// POUs/[Internal]/Beta Function Blocks/Position Correction/MC_TableBasedPositionCompensation
(*==============================================================================*)
(* Name:	MC_TableBasedPositionCompensation									*)
(*		(based on _FB_PositionCorrectionTableLookup + MC_PositionCorrectionLimiter)	*)
(* Parameter: returns a compensation value depending on the position of the reference axis	*)
(*		Use the nc function PositionCompensation to compensate a position error	*)
(*		1. the FB _FB_PositionCorrectionTableLookup calculates the correction value	*)
(*		2. the FB MC_PositionCorrectionLimiter feed this correction value		*)
(*		into the NcToPlc.PositionCorrection variable							*)
(* Author:	 	HKP																*)
(* Date:		19-July-2012													*)
(* last edit:	VER 0.0.4														*)
(*==============================================================================*)
FUNCTION_BLOCK MC_TableBasedPositionCompensation
VAR_IN_OUT
	Axis						: AXIS_REF; (*Reference to an axis*)
END_VAR
VAR_INPUT
	Enable						: BOOL; 				(* rising edge triggers initialize routine *)
	pTable						: POINTER TO ST_PositionCompensationTableElement;	(* pointer to equidistant table with strictly monotonous increasing position values *)
	TableSize					: UDINT;				(* size of data in bytes related to 'pTable' *)
	TableParameter				: ST_PositionCompensationTableParameter;(* position compensation table parameter structure *)
	Ramp						: LREAL;								(* velocity limit for feeded position compensation (constant velocity and linear position sub profile for position compensation) [mm/s] (default:=0.0) *)
	DisableMode					: E_DisableMode;						(* disable mode defines whow to react in case of disabling: (0)=HOLD, (1)=RESET, ... *)
	Options						: ST_PositionCompensationOptions;		(* optional parameters (NOT USED YET) *)
END_VAR
VAR_OUTPUT
	Enabled						: BOOL;
	Busy						: BOOL;
	Error						: BOOL;
{attribute 'displaymode':='hex'}
	ErrorID						: UDINT;
	CurrentCorrection			: LREAL;							(* current actual position correction value [mm] *)
	Limiting					: BOOL;								(* function block is currently limiting the Position Correction *)
END_VAR
VAR
	InternalEnable				: BOOL;								(* trick for internal FB handling *)
	state						: INT;
	GetThisTaskIndex			: GETCURTASKINDEX;
	CycleTime					: LREAL;							(* task cycle time [s] *)
	fbCalcPositionCorrection	: _FB_PositionCorrectionTableLookup;(* based on old 'FB_PositionCompensation' in TcNc.lib *)
	fbFeedPositionCorrection	: MC_PositionCorrectionLimiter;		(* s.TcMC2.lib (original based on old 'FB_WritePositionCorrection' in TcNc.lib) *)
	CalcPosCorrOut				: ST_McOutputs;
	FeedPosCorrOut				: ST_McOutputs;
	InternalAcceleration		: LREAL;							(* input of FB 'MC_PositionCorrectionLimiter': 'Acceleration' [mm/s^2] *)
	InternalCorrectionValue		: LREAL;							(* output of FB 'MC_PositionCorrectionLimiter': 'PositionCorrectionValue' [mm] *)
	InternalLimitingActive		: BOOL;								(* output of FB 'MC_PositionCorrectionLimiter': 'Limiting' [0/1] *)
END_VAR


CASE state OF
	0 : (* init *)
		Busy := FALSE;
		Enabled := FALSE;
		IF Enable THEN
			IF NOT Axis.NcToPlc.OpModeDWord.20 THEN (* PositionCorrection active ? *)
				Error := TRUE;
				ErrorID := MC_ERROR_WRONG_MODE;
				state := 9999;
			ELSIF Ramp < 0 THEN
				Error := TRUE;
				ErrorID := MC_ERROR_PARAMETER_NOT_CORRECT;
				state := 9999;
			ELSE
				Busy := TRUE;
				state := 1;
			END_IF
		END_IF

	1 : (* active *)
		Enabled := TRUE;


		(* cycle time needed for pre calculation of the acceleration input *)
		IF CycleTime = 0 THEN
			GetThisTaskIndex();
(*			CycleTime := SystemTaskInfoArr[GetThisTaskIndex.index].cycleTime * LREAL#100E-9;*)
			CycleTime := TwinCAT_SystemInfoVarList._TaskInfo[GetThisTaskIndex.index].cycleTime * LREAL#100E-9;
		END_IF

		(* special handling for disabling (depends from disable mode) *)
		IF( Enable = FALSE ) THEN
			(* disable mode HOLD *)
			IF( (DisableMode = DisableModeHold) ) THEN
				InternalEnable := TRUE;
				IF( Ramp > 0.0 ) THEN
					InternalAcceleration := Ramp / CycleTime;			(* mm/s^2 = mm/s / s *)
				ELSE
					InternalAcceleration := 0.0;
				END_IF
			(* disable mode RESET *)
			ELSE
				InternalEnable := Enable;
				InternalAcceleration := 0.0;
			END_IF
		(* active *)
		ELSE
			InternalEnable := Enable;
			IF( Ramp > 0.0 ) THEN
				InternalAcceleration := Ramp / CycleTime;			(* mm/s^2 = mm/s / s *)
			ELSE
				InternalAcceleration := 0.0;
			END_IF
		END_IF


		(* 1.) calculate position correction (if enabled) *)
		(* '_FB_PositionCorrectionTableLookup' *)
		fbCalcPositionCorrection(
		   (* Enable := Enable, *)
		   Enable := InternalEnable,
		   pTable := pTable,
		   TableSize := TableSize,
		   Axis := Axis,
		   TableParameter := TableParameter,
		   Compensation => InternalCorrectionValue,
		   Error => CalcPosCorrOut.Error,
		   ErrorId => CalcPosCorrOut.ErrorID,
		   Active => CalcPosCorrOut.Active );

		(* check for error return code *)
		IF CalcPosCorrOut.Error THEN
			Error := TRUE;
			ErrorID := CalcPosCorrOut.ErrorID;
			state := 9999;
		END_IF


		(* 2.) feed position compensation (acceleration limited, that means linear velocity ramp) *)
		(*
				POSITIONCORRECTIONMODE_FAST
					The limitatation to maximum position change per cycle. Due to the maximum 
					change per cycle, the correction will take place as fast as possible and may 
					also be unlimited if PositionCorrectionValue is changed slightly. 
		*)
		(* MC_PositionCorrectionLimiter *)
		fbFeedPositionCorrection(
		(*	Enable :=TRUE, *)
			 Enable :=Enable,
			 PositionCorrectionValue := InternalCorrectionValue,
			 CorrectionMode := POSITIONCORRECTION_MODE_FAST,
			 Acceleration := InternalAcceleration,			(* HKP: pre calculated internal acceleration limit *)
			 CorrectionLength := 0.0,					(* optional length - not used for this correction mode 'POSITIONCORRECTION_MODE_FAST' *)
			 Axis := Axis,
			 Busy => FeedPosCorrOut.Busy,
			 Error => FeedPosCorrOut.Error,
			 ErrorID =>FeedPosCorrOut.ErrorID,
			 Limiting => InternalLimitingActive
			);

		(* check for error return code *)
		IF FeedPosCorrOut.Error THEN
			Error := TRUE;
			ErrorID := FeedPosCorrOut.ErrorID;
			state := 9999;
		END_IF


		CurrentCorrection	:= InternalCorrectionValue;
		Limiting			:= InternalLimitingActive;

		IF NOT Enable THEN
			Enabled := FALSE;
			state := 0;
		END_IF

	9999 : (* error *)
		IF NOT Enable THEN
			Error := FALSE;
			ErrorID := 0;
			state := 0;
		END_IF
END_CASE

IF state = 0 THEN
	Busy := FALSE;
END_IF

END_FUNCTION_BLOCK

// POUs/[Internal]/_FB_PositionCorrectionTableLookup
{attribute 'conditionalshow'}
(*==========================================================================*)
(* Name:	_FB_PositionCorrectionTableLookup (based on FB_PositionCompensation)	*)
(* Parameter:	returns a compensation value depending on the position of the reference	*)
(*			axis																*)
(*																			*)
(* Author:	 	kbn & HKP														*)
(* Date:		06-July-2012														*)
(* last edit:	VER 2.0.0														*)
(*==========================================================================*)
FUNCTION_BLOCK _FB_PositionCorrectionTableLookup
VAR_IN_OUT
	Axis				: AXIS_REF; (*Reference to an axis*)
END_VAR
VAR_INPUT
	Enable			: BOOL; 				(* rising edge triggers initialize routine *)
	pTable			: POINTER TO ST_PositionCompensationTableElement;	(* pointer to table of this type *)
	TableSize		: UDINT;				(* size of data in bytes related to 'pTable' *)
	TableParameter	: ST_PositionCompensationTableParameter;	(* position compensation table parameter structure *)
END_VAR
VAR_OUTPUT
	Compensation	: LREAL;
	Error			: BOOL;
{attribute 'displaymode':='hex'}
	ErrorID			: UDINT;
	Active			: BOOL;
END_VAR
VAR
	nState			: UDINT;
	dwSize			: DWORD;
	eActiveDirection	: E_WorkDirection := WorkDirectionNone;
	bExecCalc		: BOOL;
	stElement1		: ST_PositionCompensationTableElement;
	stElement2		: ST_PositionCompensationTableElement;
	nLeftIndex		: UDINT;									(* Index starting from 0 up to (N-1) *)
	fSetPos			: LREAL;									(* position setpoint (absolute linear position or modulo position) *)
	(* HKP *)
	pTmpTable		: POINTER TO ST_PositionCompensationTableElement;	(* helper variable: pointer to table of this type *)
	fTmpStep		: LREAL;									(* helper variable *)
	fTmpA			: LREAL;									(* helper variable *)
	fTmpB			: LREAL;									(* helper variable *)
	fTmpDelta1		: LREAL;									(* helper variable *)
	fTmpDelta2		: LREAL;									(* helper variable *)
END_VAR
VAR CONSTANT
	ERRORCODE_PARAMSIZE	: UDINT := 16#4B43;
	ERRORCODE_PARAMPOS	: UDINT := 16#4B44;
(*	ERRORCODE_TCNCNOTIMPL	: UDINT := 16#4B45; *)
END_VAR

(* get last commanded direction *)
IF Axis.NcToPlc.SetVelo > 0.0001 THEN
	eActiveDirection	:= WorkDirectionPositive;
ELSIF Axis.NcToPlc.SetVelo < -0.0001 THEN
	eActiveDirection	:= WorkDirectionNegative;
END_IF

CASE nState OF
0:
	Error			:= FALSE;
	ErrorId			:= 0;
	Compensation	:= 0.0;
	Active			:= FALSE;
	bExecCalc		:= FALSE;

	IF Enable THEN
		(* reinitialize *)
		IF ( ABS(Axis.NcToPlc.SetVelo) < 0.0001 ) THEN
			eActiveDirection := WorkDirectionNone;
		END_IF
		(* check table size (in mimimum 2 elements needed) *)
		IF TableParameter.NoOfTableElements < 2 THEN
			Error	:= TRUE;
			ErrorId	:= ERRORCODE_PARAMSIZE;
			nState	:= 9999;
			RETURN;
		END_IF
		(* check table size *)
		IF TableParameter.NoOfTableElements*SIZEOF(pTable^) <> TableSize THEN
			Error	:= TRUE;
			ErrorId	:= ERRORCODE_PARAMSIZE;
			nState	:= 9999;
			RETURN;
		END_IF
		(* ====================================================== *)
		(* HKP: read table element with index (0)						*)
		(* ====================================================== *)
		(* stElement1	:= F_GetCompensationElementAt(pTable:=pTable, nElement:=0); *)
		pTmpTable	:= pTable + (SIZEOF(pTable^) * (UDINT#0));
		stElement1	:= pTmpTable^;
		(* ====================================================== *)
		IF stElement1.Position <> TableParameter.MinPosition THEN
			Error	:= TRUE;
			ErrorId	:= ERRORCODE_PARAMPOS;
			nState	:= 9999;
			RETURN;
		END_IF
		(* ====================================================== *)
		(* HKP: read table element with index (Parameter.nTableElements-1)	*)
		(* ====================================================== *)
		(* stElement1	:= F_GetCompensationElementAt(pTable:=pTable, nElement:=Parameter.nTableElements-1); *)
		pTmpTable	:= pTable + (SIZEOF(pTable^) * (TableParameter.NoOfTableElements-1));
		stElement1	:= pTmpTable^;
		(* ====================================================== *)
		IF stElement1.Position <> TableParameter.MaxPosition THEN
			Error	:= TRUE;
			ErrorId	:= ERRORCODE_PARAMPOS;
			nState	:= 9999;
			RETURN;
		END_IF
		(* HKP: This two parameter are not needed yet *)
		(* IF Parameter.eTableType <> TableType1DEquidistant OR Parameter.bModulo THEN
			Error	:= TRUE;
			ErrorId	:= ERRORCODE_TCNCNOTIMPL;
			nState	:= 9999;
			RETURN;
		END_IF *)

		(* check for equidistant table (table must contain in minimum 2 elements) *)
		pTmpTable	:= pTable + (SIZEOF(pTable^) * (UDINT#1));						(* read index 1 *)
		stElement2	:= pTmpTable^;
		pTmpTable	:= pTable + (SIZEOF(pTable^) * (UDINT#0));						(* read index 0 *)
		stElement1	:= pTmpTable^;
		fTmpDelta1	:= stElement2.Position - stElement1.Position;						(* calculate position delta 1: (index 1 - index 0) *)
		pTmpTable	:= pTable + (SIZEOF(pTable^) * (TableParameter.NoOfTableElements-1));	(* read index (n) *)
		stElement2	:= pTmpTable^;
		pTmpTable	:= pTable + (SIZEOF(pTable^) * (TableParameter.NoOfTableElements-2));	(* read index (n-1) *)
		stElement1	:= pTmpTable^;
		fTmpDelta2	:= stElement2.Position - stElement1.Position;						(* calculate position delta 2: (index (n) - index (n-1)) *)
		IF( ABS(fTmpDelta2 - fTmpDelta1) > 1.0E-6 ) THEN
			Error	:= TRUE;
			ErrorId	:= ERRORCODE_PARAMPOS;
			nState	:= 9999;
			RETURN;
		END_IF

		(* ====================================================== *)
		(* HKP: call action 'F_IsCompensationDirection()'				*)
		(* INPUT: eActive:=eActiveDirection, eRequested:=Parameter.Direction *)
		(* OUTPUT: bExecCalc									*)
		(* ====================================================== *)
		(* bExecCalc	:= F_IsCompensationDirection(eActive:=eActiveDirection, eRequested:=Parameter.Direction); *)
		ActIsCompensationDirection( );
		(* ====================================================== *)
		nState	:= 10;
	END_IF
10:
	(* ====================================================== *)
	(* HKP: call action 'F_IsCompensationDirection()'				*)
	(* INPUT: eActive:=eActiveDirection, eRequested:=Parameter.Direction *)
	(* OUTPUT: bExecCalc									*)
	(* ====================================================== *)
	(* bExecCalc	:= F_IsCompensationDirection(eActive:=eActiveDirection, eRequested:=Parameter.Direction); *)
	ActIsCompensationDirection( );
	(* ====================================================== *)
	IF NOT Enable THEN
		bExecCalc	:= FALSE;
		nState		:= 0;
	END_IF


9999:
	IF NOT Enable THEN
		nState	:= 0;
	END_IF

END_CASE


IF bExecCalc THEN
	(* compensation is generally enabled & direction is ok *)
	Active	:= TRUE;
	(* modulo or linear axis? *)
	IF( TableParameter.Modulo )THEN
		fSetPos	:= Axis.NcToPlc.ModuloSetPos;
	ELSE
		fSetPos	:= Axis.NcToPlc.SetPos;
	END_IF
	IF fSetPos < TableParameter.MinPosition THEN
		(* ====================================================== *)
		(* HKP: read table element with index (0)						*)
		(* ====================================================== *)
		(* stElement1	:= F_GetCompensationElementAt(pTable:=pTable, nElement:=0 ); *)
		pTmpTable	:= pTable + (SIZEOF(pTable^) * (UDINT#0));
		stElement1	:= pTmpTable^;
		(* ====================================================== *)
		Compensation	:= stElement1.Compensation;
	ELSIF fSetPos > TableParameter.MaxPosition THEN
		(* ====================================================== *)
		(* HKP: read table element with index (Parameter.nTableElements-1)	*)
		(* ====================================================== *)
		(* stElement1	:= F_GetCompensationElementAt(pTable:=pTable, nElement:=Parameter.nTableElements-1); *)
		pTmpTable	:= pTable + (SIZEOF(pTable^) * (TableParameter.NoOfTableElements-1));
		stElement1	:= pTmpTable^;
		(* ====================================================== *)
		Compensation := stElement1.Compensation;
	ELSE
		(* ====================================================== *)
		(* HKP: get left table index to position (Axis.NcToPlc.SetPos)		*)
		(* ====================================================== *)
		(* nLeftIndex	:= F_GetLeftIndex(fPos:=Axis.NcToPlc.SetPos, fMin:=Parameter.MinPosition, fMax:=Parameter.MaxPosition, nCount:=Parameter.NoOfTableElements); *)
		IF TableParameter.NoOfTableElements <= 1 THEN
			nLeftIndex := 0;
		ELSE
			IF fSetPos < TableParameter.MinPosition THEN
				nLeftIndex	:= 0;
			ELSIF fSetPos > TableParameter.MaxPosition THEN
				nLeftIndex	:= TableParameter.NoOfTableElements-1;
			ELSE
				fTmpStep	:= (TableParameter.MaxPosition-TableParameter.MinPosition)/UDINT_TO_LREAL(TableParameter.NoOfTableElements-1);
				nLeftIndex	:= LREAL_TO_UDINT(FLOOR((fSetPos-TableParameter.MinPosition)/fTmpStep));
			END_IF
		END_IF
		(* ====================================================== *)
		IF nLeftIndex >= TableParameter.NoOfTableElements-1 THEN
			(* there is no right index - probably fPos is exactly 'MaxPosition' *)
			(* ====================================================== *)
			(* HKP: read table element with index (Parameter.nTableElements-1)	*)
			(* ====================================================== *)
			(* stElement1	:= F_GetCompensationElementAt(pTable:=pTable, nElement:=Parameter.nTableElements-1); *)
			pTmpTable	:= pTable + (SIZEOF(pTable^) * (TableParameter.NoOfTableElements-1));
			stElement1	:= pTmpTable^;
			(* ====================================================== *)
			Compensation	:= stElement1.Compensation;
		ELSE
			(* ====================================================== *)
			(* HKP: read table element with index (nLeftIndex)				*)
			(* HKP: read table element with index (nLeftIndex+1)				*)
			(* ====================================================== *)
			(* stElement1	:= F_GetCompensationElementAt(pTable:=pTable, nElement:=nLeftIndex); *)
			(* stElement2	:= F_GetCompensationElementAt(pTable:=pTable, nElement:=nLeftIndex+1); *)
			pTmpTable	:= pTable + (SIZEOF(pTable^) * nLeftIndex);
			stElement1	:= pTmpTable^;
			pTmpTable	:= pTable + (SIZEOF(pTable^) * (nLeftIndex+1));
			stElement2	:= pTmpTable^;
			(* ====================================================== *)
			(* ====================================================== *)
			(* HKP: calculate linear interpolation between (stElement1) and (stElement2) for position (Axis.NcToPlc.SetPos)	*)
			(* ====================================================== *)
			(* Compensation	:= F_LinearInterpolationCompensation(fPos:=Axis.NcToPlc.SetPos, stElement1:=stElement1, stElement2:=stElement2); *)
			(* y := ax+b*)
			(* a:=(y2-y1)/(x2-x1)*)
			fTmpA	:= (stElement2.Compensation-stElement1.Compensation) / (stElement2.Position-stElement1.Position);
			(* b:=y-ax1 *)
			fTmpB	:= stElement1.Compensation - fTmpA*stElement1.Position;
			Compensation := fTmpA*fSetPos + fTmpB;
			(* ====================================================== *)
		END_IF
	END_IF
ELSE
	Compensation	:= 0.0;
	Active			:= FALSE;
END_IF

ACTION ActIsCompensationDirection:
(*
FUNCTION F_IsCompensationDirection : BOOL
VAR_INPUT
	eActiveDirection		: E_WorkingDirection;	( eActive		: E_WorkingDirection )
	Parameter.Direction	: E_WorkingDirection;	( eRequested	: E_WorkingDirection )
END_VAR
VAR_OUTPUT
	bExecCalc		: BOOL;				( F_IsCompensationDirection : BOOL )
END_VAR
*)

(*
         |Active |       |       |       |
         |None   | both  | plus  | minus |
---------|-------|-------|-------|-------|
Req None |  0    |  0    |  0    |  0    |
---------|-------|-------|-------|-------|
Req both |  1    |  d.c. |  1    |  1    |
---------|-------|-------|-------|-------|
Req plus |  0    |  0    |  1    |  0    |
---------|-------|-------|-------|-------|
Req minus|  0    |  0    |  0    |  1    |
---------|-------|-------|-------|-------|

d.c.= don't care
*)

IF TableParameter.Direction = WorkDirectionBoth THEN
	bExecCalc	:= TRUE;
	RETURN;
END_IF
IF eActiveDirection = WorkDirectionPositive AND TableParameter.Direction = WorkDirectionPositive  THEN
	bExecCalc	:= TRUE;
	RETURN;
END_IF
IF eActiveDirection = WorkDirectionNegative AND TableParameter.Direction = WorkDirectionNegative  THEN
	bExecCalc	:= TRUE;
	RETURN;
END_IF
bExecCalc		:= FALSE;


(*
IF eActiveDirection = WorkingDirectionPlus AND (TableParameter.Direction = WorkingDirectionBoth OR TableParameter.Direction = WorkingDirectionPlus ) THEN
	bExecCalc	:= TRUE;
	RETURN;
END_IF
IF eActiveDirection = WorkingDirectionMinus AND (TableParameter.Direction = WorkingDirectionBoth OR TableParameter.Direction = WorkingDirectionMinus ) THEN
	bExecCalc	:= TRUE;
	RETURN;
END_IF
bExecCalc		:= FALSE;
*)
END_ACTION

END_FUNCTION_BLOCK

// POUs/Administrative/Extensions/MC_PositionCorrectionLimiter
FUNCTION_BLOCK MC_PositionCorrectionLimiter
(*
 	The function block PositionCorrectionLimiter feed a correction value into the
	NcToPlc.PositionCorrection variable. 

	The correction value corrects the actual position of the encoder. The correction 
	does not only affect the actual position but will also lead to an axis motion caused 
	by the position controller of the axis or drive. The correction does not affect the
	set position of the set-point generator.

	The block supports following modes:
		POSITIONCORRECTIONMODE_UNLIMITED
			no limitation - the PositionCorrectionValue is passed to the NC immediately
		POSITIONCORRECTIONMODE_FAST
			The limitatation to maximum position change per cycle. Due to the maximum 
			change per cycle, the correction will take place as fast as possible and may 
			also be unlimited if PositionCorrectionValue is changed slightly. 
		POSITIONCORRECTIONMODE_FULLLENGTH 
			The limitation uses a defined full CorrectionLength (travel path)  to adapt to 
			the PositionCorrectionValue in small steps. This mode will allways cause a 
			limitation and takes care of a smooth correction.
*)
VAR_IN_OUT
	Axis					:	AXIS_REF; (*Reference to an axis*)
END_VAR
VAR_INPUT
	Enable				:	BOOL;
	PositionCorrectionValue : 	LREAL;
	CorrectionMode		:	E_AxisPositionCorrectionMode;
	Acceleration			: 	LREAL;
	CorrectionLength		:	LREAL; (* optional length - comparable to 'superposition length' *)
END_VAR
VAR_OUTPUT
	Busy				:	BOOL;
	Error				:	BOOL;
{attribute 'displaymode':='hex'}
	ErrorID				:	UDINT;
	Limiting				: 	BOOL;	(* function block is currently limiting the Position Correction *)
END_VAR
VAR
	GetThisTaskIndex: GETCURTASKINDEX;
	CycleTime: LREAL;
	MaxDeltaVelocity: LREAL;
	MaxDeltaPosition: LREAL;
	DeltaCorrection: LREAL;
	InitialDeltaCorrection: LREAL;
	EndOfEnablePhase: BOOL;
	iCorrectionMode : E_AxisPositionCorrectionMode;
	state: INT;
	NumberOfCycles: UDINT;
	DeltaCorrectionPerCycle: LREAL;
	LastPositionCorrectionValue: LREAL;
	LastPositionCorrection: LREAL;
END_VAR

CASE state OF
	0 : (* disabled *)
		Busy := FALSE;
		Limiting := FALSE;
		LastPositionCorrectionValue := 0;
		IF Enable THEN
			(* IF Acceleration<=0 AND CorrectionMode <> POSITIONCORRECTION_MODE_UNLIMITED THEN *) (* KST 20120730 *)
			IF Acceleration<0 AND CorrectionMode <> POSITIONCORRECTION_MODE_UNLIMITED THEN (* KST 20120730 - zero acc means unlimited correction *)
				Error := TRUE;
				ErrorID := MC_ERROR_PARAMETER_NOT_CORRECT;
			ELSIF CorrectionLength <= 0 AND CorrectionMode=POSITIONCORRECTION_MODE_FULLLENGTH THEN
				Error := TRUE;
				ErrorID := MC_ERROR_PARAMETER_NOT_CORRECT;
			ELSE
				Limiting := FALSE;
				Error := FALSE;
				ErrorID := 0;
				LastPositionCorrection := Axis.PlcToNc.PositionCorrection; // KST 2021-02-23 store position correction value
				state := 1;
				Busy := TRUE;
			END_IF
		ELSE
			Limiting := FALSE;
			Error := FALSE;
			ErrorID := 0;
		END_IF

	1 : (* enabled *)
		Busy := TRUE;
		IF NOT Enable THEN
			state := 2;
		END_IF

	2 : (* disabling *)
		IF Enable THEN
			LastPositionCorrection := Axis.PlcToNc.PositionCorrection; // KST 2021-09-27 store position correction value
			state := 1;
		ELSE
			PositionCorrectionValue := 0;
//			IF Axis.PlcToNc.PositionCorrection = 0 THEN
			IF LastPositionCorrection = 0 THEN	// KST 2021-02-23
				state := 0;
			END_IF
		END_IF
END_CASE

CASE state OF
	1, 2:
		IF CycleTime = 0 THEN
			GetThisTaskIndex();
			CycleTime := TwinCAT_SystemInfoVarList._TaskInfo[GetThisTaskIndex.index].cycleTime * LREAL#100E-9;
		END_IF
		MaxDeltaVelocity := Acceleration * CycleTime;
		MaxDeltaPosition := MaxDeltaVelocity * CycleTime;
//		DeltaCorrection := PositionCorrectionValue - Axis.PlcToNc.PositionCorrection;
		DeltaCorrection := PositionCorrectionValue - LastPositionCorrection;	// KST 2021-02-23
		
		(* check if correction mode is possible *)
		iCorrectionMode := CorrectionMode;
		
(*		IF iCorrectionMode=POSITIONCORRECTION_MODE_FULLLENGTH AND CorrectionLength <= 0 OR ABS(Axis.NcToPlc.SetVelo) < 1E-6 THEN*)	(* KSt 2013-09-02 brackets wrong *)
		IF iCorrectionMode=POSITIONCORRECTION_MODE_FULLLENGTH AND (CorrectionLength <= 0 OR ABS(Axis.NcToPlc.SetVelo) < 1E-6) THEN	(* KSt 2013-09-02 brackets new *)
			iCorrectionMode := POSITIONCORRECTION_MODE_FAST;
		END_IF

		CASE iCorrectionMode OF
			POSITIONCORRECTION_MODE_UNLIMITED :
					Limiting := FALSE;
					Axis.PlcToNc.PositionCorrection := PositionCorrectionValue;

			POSITIONCORRECTION_MODE_FAST :
				(* IF ABS(DeltaCorrection) <= MaxDeltaPosition then *) (* KST 20120730 *)
				IF 	ABS(DeltaCorrection) <= MaxDeltaPosition
					OR Acceleration=0 OR MaxDeltaPosition=0 (* KST 20120730 - zero acc means unlimited correction *)
					THEN
					Limiting := FALSE;
					Axis.PlcToNc.PositionCorrection := PositionCorrectionValue;
				ELSE
					Limiting := TRUE;
					IF DeltaCorrection > 0 THEN
//						Axis.PlcToNc.PositionCorrection := Axis.PlcToNc.PositionCorrection + MaxDeltaPosition;
						Axis.PlcToNc.PositionCorrection := LastPositionCorrection + MaxDeltaPosition;	// KST 2021-02-23
					ELSE
//						Axis.PlcToNc.PositionCorrection := Axis.PlcToNc.PositionCorrection - MaxDeltaPosition;
						Axis.PlcToNc.PositionCorrection := LastPositionCorrection - MaxDeltaPosition;	// KST 2021-02-23
					END_IF
				END_IF

			POSITIONCORRECTION_MODE_FULLLENGTH :
				(* check if PositionCorrectionValue changed *)
				(* then calculate the change per cycle and scatter the change over the defined CorrectionLength *)
				IF PositionCorrectionValue<>LastPositionCorrectionValue THEN
					InitialDeltaCorrection := DeltaCorrection;
				END_IF
				LastPositionCorrectionValue := PositionCorrectionValue;
				NumberOfCycles := LREAL_TO_UDINT(CorrectionLength / ABS(Axis.NcToPlc.SetVelo) / CycleTime);
				NumberOfCycles := MAX(NumberOfCycles,1);	// KSt 2021-11-11   avoid zero division 
				DeltaCorrectionPerCycle := ABS(InitialDeltaCorrection) / NumberOfCycles;
(*				IF ABS(DeltaCorrectionPerCycle) > MaxDeltaPosition THEN*) (* KST 20120730 *)
				IF 	ABS(DeltaCorrectionPerCycle) > MaxDeltaPosition
					AND MaxDeltaPosition > 0 THEN (* KST 20120730 *)
					DeltaCorrectionPerCycle := MaxDeltaPosition;
				END_IF

				IF ABS(DeltaCorrection) <= DeltaCorrectionPerCycle THEN
					Limiting := FALSE;
					Axis.PlcToNc.PositionCorrection := PositionCorrectionValue;
				ELSE
					Limiting := TRUE;
					IF DeltaCorrection > 0 THEN
//						Axis.PlcToNc.PositionCorrection := Axis.PlcToNc.PositionCorrection + DeltaCorrectionPerCycle;
						Axis.PlcToNc.PositionCorrection := LastPositionCorrection + DeltaCorrectionPerCycle;	// KST 2021-02-23
					ELSE
//						Axis.PlcToNc.PositionCorrection := Axis.PlcToNc.PositionCorrection - DeltaCorrectionPerCycle;
						Axis.PlcToNc.PositionCorrection := LastPositionCorrection - DeltaCorrectionPerCycle;	// KST 2021-02-23
					END_IF
				END_IF
		END_CASE
		LastPositionCorrection := Axis.PlcToNc.PositionCorrection; // KST 2021-02-23 store position correction value
END_CASE

END_FUNCTION_BLOCK

// POUs/[Internal]/Beta Function Blocks/Sinus motion/MC_SinusOscillation
FUNCTION_BLOCK MC_SinusOscillation
VAR_IN_OUT
	Axis			:	AXIS_REF; (*Reference to an axis*)
END_VAR
VAR_INPUT
	Execute			:	BOOL;
	VeloAmplitude	:	LREAL;
	Frequency		:	LREAL;
	DrivingTime		:	TIME;
END_VAR
VAR_OUTPUT
	Busy			:	BOOL;
	Active			:	BOOL;
	Done			:	BOOL;
	Error			:	BOOL;
{attribute 'displaymode':='hex'}
	ErrorID			:	UDINT;
END_VAR
VAR
	_FB_MoveSinusGeneric	: _FB_MoveSinusGeneric;
END_VAR

_FB_MoveSinusGeneric.stData.StartType 					:= 0;
_FB_MoveSinusGeneric.stData.BaseAmplitude				:= 2.5; // fixed value
_FB_MoveSinusGeneric.stData.BaseFrequency				:= 1.953125; // fixed value
_FB_MoveSinusGeneric.stData.StartAmplitudeAtBeginn		:= VeloAmplitude;
_FB_MoveSinusGeneric.stData.FeedConstantMotor			:= 10.0; // fixed value
_FB_MoveSinusGeneric.stData.StartFrequency				:= Frequency;
_FB_MoveSinusGeneric.stData.StopFrequency				:= 500.0; // fixed value
_FB_MoveSinusGeneric.stData.StepDuration				:= TIME_TO_LREAL(DrivingTime)/1000;
_FB_MoveSinusGeneric.stData.NumberMeasurements			:= 1;
_FB_MoveSinusGeneric.stData.NumberParallelMeasurements	:= 0;

_FB_MoveSinusGeneric(
	Axis				:= Axis, 
	Execute				:= Execute, 
	Mode				:= _E_SinusMotionMode.eSinusMode_Oscillation, 
	stData				:= , 
	Busy				=> Busy, 
	Active				=> Active, 
	Done				=> Done, 
	Error				=> Error, 
	ErrorID				=> ErrorId);

END_FUNCTION_BLOCK

// POUs/[Internal]/_FB_MoveSinusGeneric
{attribute 'conditionalshow'}
FUNCTION_BLOCK _FB_MoveSinusGeneric
VAR_IN_OUT
	Axis			: AXIS_REF; (*Reference to an axis*)
END_VAR
VAR_INPUT
	Execute			: BOOL;
	Mode			: _E_SinusMotionMode;
	stData			: _ST_TcNc_SinusMotion;
END_VAR
VAR_OUTPUT
	Busy			: BOOL;
	Active			: BOOL;
	Done			: BOOL;
	Error			: BOOL;
{attribute 'displaymode':='hex'}
	ErrorID			: UDINT;
END_VAR
VAR
	GetTaskIndex	: GETCURTASKINDEX;
	CycleTime		: LREAL;								(* task cycle time [s] *)
	fbAdsWrite		: ADSWRITE;// := ( NETID := Axis.ADS.NetId, PORT := Axis.ADS.Port, TMOUT := DEFAULT_ADS_TIMEOUT );
	fbOnTrigger		: R_Trig;
	nState			: _E_TcMC_STATES;
	Info: LREAL;
END_VAR

(*---------------------- Rising/Falling Edge Detection ----------------------*)
fbOnTrigger(CLK:= Execute);

(*---------------------- State Machine ----------------------*)
CASE nState OF
	STATE_INITIALIZATION:	// Initialisation
		Busy	:= FALSE;
		Active	:= FALSE;
		IF NOT Execute THEN			// reset at falling edge of Execute
			Done 	:= FALSE;
			Error 	:= FALSE;
			ErrorID := 0;
		END_IF

		fbAdsWrite(	WRITE := FALSE ); // Write auf False setzen, damit es später eine steigende Flanke gibt!
		
		IF fbOnTrigger.Q THEN
			(*---------------------- Writing Data into Structure ----------------------*)
			IF CycleTime = 0 THEN
				GetTaskIndex();
				CycleTime := TwinCAT_SystemInfoVarList._TaskInfo[GetTaskIndex.index].cycleTime * LREAL#100E-9;
			END_IF

			stData.StartType					:= 0;			// Not Used Yet!
			CASE Mode OF
				_E_SinusMotionMode.eSinusMode_Oscillation:
					IF stData.StartAmplitudeAtBeginn <= 0.0 THEN										// Check Parameter in Wertebereich
						Error := 1;
						ErrorID := E_AxisErrorCodes.MC_ERROR_PARAMETER_NOT_CORRECT;
					END_IF
					IF stData.StartFrequency <= 0.0 OR stData.StartFrequency > (1/(2*CycleTime)) THEN	// Check Parameter in Wertebereich
						Error := 1;
						ErrorID := E_AxisErrorCodes.MC_ERROR_PARAMETER_NOT_CORRECT;
					END_IF
			
				_E_SinusMotionMode.eSinusMode_Sequence:
					IF stData.BaseAmplitude <= 0.0 THEN													// Check Parameter in Wertebereich
						Error := 1;
						ErrorID := E_AxisErrorCodes.MC_ERROR_PARAMETER_NOT_CORRECT;
					END_IF
					IF stData.FeedConstantMotor <= 0.0 THEN												// Check Parameter in Wertebereich
						Error := 1;
						ErrorID := E_AxisErrorCodes.MC_ERROR_PARAMETER_NOT_CORRECT;
					END_IF
					IF stData.StartFrequency < 1.0 OR stData.StartFrequency > (1/(2* CycleTime)) THEN	// Check Parameter in Wertebereich
						Error := 1;
						ErrorID := E_AxisErrorCodes.MC_ERROR_PARAMETER_NOT_CORRECT;
					END_IF
					IF stData.StopFrequency < 1.0 OR stData.StopFrequency > (1/(2*CycleTime)) THEN		// Check Parameter in Wertebereich
						Error := 1;
						ErrorID := E_AxisErrorCodes.MC_ERROR_PARAMETER_NOT_CORRECT;
					END_IF
					IF stData.BaseFrequency < 0.0 OR stData.BaseFrequency > 10.0 OR stData.BaseFrequency > (1/(2*CycleTime)) THEN		// Check Parameter in Wertebereich
						Error := 1;
						ErrorID := E_AxisErrorCodes.MC_ERROR_PARAMETER_NOT_CORRECT;
					END_IF
					IF stData.StopFrequency < stData.StartFrequency THEN								// Check if StopFrequency is larger than StartFrequency
						Error := 1;
						ErrorID := E_AxisErrorCodes.MC_ERROR_PARAMETER_NOT_CORRECT;
					END_IF								
					IF stData.NumberMeasurements < 1 OR stData.NumberMeasurements > 200 THEN			// Check Parameter in Wertebereich
						Error := 1;
						ErrorID := E_AxisErrorCodes.MC_ERROR_PARAMETER_NOT_CORRECT;
					END_IF
			END_CASE
			IF stData.StepDuration <= 0.0 THEN													// Check Parameter in Wertebereich
				Error := 1;
				ErrorID := E_AxisErrorCodes.MC_ERROR_PARAMETER_NOT_CORRECT;
			END_IF

			(*---------------------- Checking for Erros before ADS write to start Axis ----------------------*)
			IF Error THEN
				nState := STATE_INITIALIZATION;
			ELSE
				Busy 	:= TRUE;
				Active	:= FALSE;
				Done 	:= FALSE;
				nState 	:= STATE_ORDER;
				
				fbAdsWrite(
					NETID		:= '',							//Axis.ADS.NetId,
					PORT		:= AMSPORT_R0_NCSAF,			//Axis.ADS.Port, 
					IDXGRP		:= 16#4200+Axis.NcToPlc.AxisId, // Index-Gruppennummer (0x4200+Axis.NcToPlc.AxisId) des Dienstes 
					IDXOFFS		:= 16#33, 						// Index-Offsetnummer (0x00000033) des Dienstes (Sinus Oscillation)
					LEN			:= SIZEOF(stData),				// Länge der zu übergebenden Struktur
					SRCADDR		:= ADR(stData),					// Adresse der Struktur
					WRITE		:= TRUE, 						// Steigende Flanke für Schreiben des Befehls!
					TMOUT		:= DEFAULT_ADS_TIMEOUT,			// Timeout, nachdem der Befehl abgebrochen wird (5s)
					BUSY		=> , 
					ERR			=> , 
					ERRID		=> );
			END_IF
		END_IF
		
	//-------------------------
	STATE_ORDER:	// Write Command to ADS

		fbAdsWrite();
		IF NOT fbAdsWrite.Busy THEN					// Wait until ADSwrite is not working any more
			IF fbAdsWrite.Err THEN
				Error 	:= TRUE;
				ErrorID := fbAdsWrite.ErrId;
				nState 	:= STATE_INITIALIZATION;	// Error
			ELSE 
				nState 	:= STATE_RUNNING;
			END_IF
		END_IF
	
	//-------------------------
	STATE_RUNNING:	// Sinusoidal Movement of the Axis until standstill
		
		IF Axis.NcToPlc.StateDWord.31 THEN		// AxisError
			Error 	:= TRUE;
			ErrorID := Axis.NcToPlc.ErrorCode;
			nState 	:= STATE_INITIALIZATION;	// Error
		END_IF
		
		IF Axis.NcToPlc.StateDWord.8 AND NOT Axis.NcToPlc.StateDWord.2 THEN		// AxisHasJob AND NOT NOTMoving
			Busy	:= TRUE;
			Active 	:= TRUE;
			Done	:= FALSE;
		END_IF
		
		IF NOT Axis.NcToPlc.StateDWord.8 AND Axis.NcToPlc.StateDWord.2 THEN		// NOT AxisHasJob AND NOTMoving
			Busy	:= TRUE;
			Active	:= FALSE;
			Done	:= TRUE;
			nState 	:= STATE_INITIALIZATION;
		END_IF
	
END_CASE

END_FUNCTION_BLOCK

// POUs/[Internal]/Beta Function Blocks/Sinus motion/MC_SinusSequence
FUNCTION_BLOCK MC_SinusSequence
VAR_IN_OUT
	Axis			:	AXIS_REF; (*Reference to an axis*)
END_VAR
VAR_INPUT
	Execute				: BOOL;
	StartFrequency		: LREAL;
	StopFrequency		: LREAL;
	BaseFrequency		: LREAL := 1.953125;
	FrequencySteps		: UINT;
	SinusBaseVelocity 	: LREAL;
	StepDuration		: TIME;
	FeedConstantMotor	: LREAL;
END_VAR
VAR_OUTPUT
	Busy			:	BOOL;
	Active			:	BOOL;
	Done			:	BOOL;
	Error			:	BOOL;
{attribute 'displaymode':='hex'}
	ErrorID			:	UDINT;
END_VAR
VAR
	_FB_MoveSinusGeneric	: _FB_MoveSinusGeneric;
END_VAR

_FB_MoveSinusGeneric.stData.StartType 					:= 0;
_FB_MoveSinusGeneric.stData.BaseAmplitude				:= SinusBaseVelocity;
_FB_MoveSinusGeneric.stData.BaseFrequency				:= BaseFrequency;
_FB_MoveSinusGeneric.stData.StartAmplitudeAtBeginn		:= 0.0;			// BODE-PLOT!!!
_FB_MoveSinusGeneric.stData.FeedConstantMotor			:= FeedConstantMotor;
_FB_MoveSinusGeneric.stData.StartFrequency				:= StartFrequency;
_FB_MoveSinusGeneric.stData.StopFrequency				:= StopFrequency;
_FB_MoveSinusGeneric.stData.StepDuration				:= TIME_TO_LREAL(StepDuration)/1000;
_FB_MoveSinusGeneric.stData.NumberMeasurements			:= FrequencySteps;
_FB_MoveSinusGeneric.stData.NumberParallelMeasurements	:= 1;

_FB_MoveSinusGeneric(
	Axis				:= Axis, 
	Execute				:= Execute, 
	Mode				:= _E_SinusMotionMode.eSinusMode_Sequence, 
	stData				:= , 
	Busy				=> Busy, 
	Active				=> Active, 
	Done				=> Done, 
	Error				=> Error, 
	ErrorID				=> ErrorId);

END_FUNCTION_BLOCK

// POUs/[Internal]/Beta Function Blocks/MC_ReadApplicationRequest
FUNCTION_BLOCK MC_ReadApplicationRequest
(*	This Function Block returns a data set containing all parameters of an application request *)
VAR_IN_OUT
	ApplicationRequest 	: 	ST_NcApplicationRequest;
	Axis			:	AXIS_REF; (*Reference to an axis*)
END_VAR
VAR_INPUT
	Execute		: 	BOOL;
END_VAR
VAR_OUTPUT
	Done 		: 	BOOL;
	Busy		: 	BOOL;
	Error 		: 	BOOL;
{attribute 'displaymode':='hex'}
	ErrorID 		: 	UDINT;
	Request		: 	BOOL;		(* application request bit [0/1] *)
	RequestType	: 	UINT;		(* application request TYPE/ID *)
END_VAR
VAR
	TriggerExecute: R_TRIG;
	state: _E_TcMC_STATES := STATE_INITIALIZATION;
	fbAdsRead		: 	ADSREAD;
END_VAR

TriggerExecute(CLK:=Execute);

CASE state OF
	STATE_INITIALIZATION:
		IF NOT Execute THEN
			Done := FALSE;
			Error := FALSE;	(* reset at falling edge of Execute *)
			ErrorID := 0;
		END_IF
		IF TriggerExecute.Q THEN
			Done := FALSE;
			Busy := TRUE;
			Error := FALSE;
			ErrorID := 0;
			Request := FALSE;
			RequestType := 0 ;
			fbAdsRead(READ:=FALSE);
		END_IF
		IF Busy THEN
			fbAdsRead(
				NETID:= TcMcGlobal.NCNETID_TCMC,
				PORT:= TcMcGlobal.NCPORT_TCMC,
				IDXGRP:=TcMcGlobal.Axis.Parameter.IDXGRP+Axis.NcToPlc.AxisId,
				IDXOFFS:= TcMcGlobal.Axis.Parameter.IDXOFFS.APPLICATIONREQUEST,
				LEN:= SIZEOF(ApplicationRequest),
				DESTADDR:= ADR(ApplicationRequest),
				READ:= TRUE,
				TMOUT:= TcMcGlobal.tADSTimeOut );
			IF NOT fbAdsRead.BUSY THEN
				Error := fbAdsRead.ERR;
				ErrorID := fbAdsRead.ERRID;
				Done := NOT Error;
				IF Done THEN
					Request := ApplicationRequest.bApplRequestBit<>0;
					RequestType := ApplicationRequest.nApplRequestType;
				END_IF
				Busy := FALSE;
			END_IF
		END_IF
END_CASE

END_FUNCTION_BLOCK

// POUs/[Internal]/Beta Function Blocks/MC_ReadStopInfo
FUNCTION_BLOCK MC_ReadStopInfo
(*	This Function Block returns time and distance that is required
	to stop an axis from its current dynamical state using the 
	parameterized deceleration and jerk values.
	(No motion is actually commanded by this funciton block)
*)
VAR_IN_OUT
	Axis				:	AXIS_REF; (*Reference to an axis*)
END_VAR
VAR_INPUT
	Execute			:	BOOL;	(* B *)
	Deceleration		:	LREAL;	(* E *)
	Jerk				:	LREAL;	(* E *)
END_VAR
VAR_OUTPUT
	Done 		: 	BOOL;	(* B *)
	Busy		: 	BOOL;	(* E *)
	Error 		: 	BOOL;	(* B *)
{attribute 'displaymode':='hex'}
	ErrorID 		: 	UDINT;	(* E *)
	StopDistance : 	LREAL;	(* distance required to stop the axis *)
	StopTime	: 	LREAL;	(* time required to stop the axis *)
END_VAR
VAR
	TriggerExecute: R_TRIG;
	state: _E_TcMC_STATES := STATE_INITIALIZATION;
	stStopInfoRequest 	: 	_ST_TcNC_StopInfoRequest;
	stStopInfoResponse 	: 	_ST_TcNC_StopInfoResponse;
	fbAdsReadWrite		: 	ADSRDWRT;
END_VAR

TriggerExecute(CLK:=Execute);

CASE state OF
	STATE_INITIALIZATION:
		IF NOT Execute THEN
			Done := FALSE;
			Error := FALSE;	(* reset at falling edge of Execute *)
			ErrorID := 0;
		END_IF
		IF TriggerExecute.Q THEN
			Done := FALSE;
			Busy := TRUE;
			Error := FALSE;
			ErrorID := 0;
			StopDistance := 0 ;
			StopTime := 0 ;
			stStopInfoRequest.Deceleration := Deceleration;
			stStopInfoRequest.Jerk := Jerk;
			fbAdsReadWrite(WRTRD:=FALSE);
		END_IF
		IF Busy THEN

			fbAdsReadWrite(
				NETID:= TcMcGlobal.NCNETID_TCMC,
				(*PORT:= TcMcGlobal.NCPORT_TCMC,*)
				(* FAP 2019-12-12 Changed to NCSAF port 501 to have deterministic responses *)
				PORT:= AMSPORT_R0_NCSAF, 
				IDXGRP:=TcMcGlobal.Axis.State.IDXGRP+Axis.NcToPlc.AxisId,
				IDXOFFS:= TcMcGlobal.Axis.State.IDXOFFS.STOPINFORMATION,
				WRITELEN:= SIZEOF(stStopInfoRequest),
				READLEN:= SIZEOF(stStopInfoResponse),
				SRCADDR:= ADR(stStopInfoRequest),
				DESTADDR:= ADR(stStopInfoResponse),
				WRTRD:= TRUE,
				TMOUT:= TcMcGlobal.tADSTimeOut );
			IF NOT fbAdsReadWrite.BUSY THEN
				Error := fbAdsReadWrite.ERR;
				ErrorID := fbAdsReadWrite.ERRID;
				Done := NOT Error;
				IF Done THEN
					StopDistance := stStopInfoResponse.StopDistance;
					StopTime := stStopInfoResponse.StopTime;
				END_IF
				Busy := FALSE;
			END_IF
		END_IF
END_CASE

END_FUNCTION_BLOCK

// POUs/[Internal]/Objects/_TCMCGLOBAL
(*	Global constants and parameters *)
{attribute 'conditionalshow'}
FUNCTION_BLOCK _TCMCGLOBAL
VAR_INPUT
	NCPORT_TCMC 				: UINT 	:= AMSPORT_R0_NC;  (* 20110511 type changed from INT to UINT *)
	NCPORT_TCMC_COUPLING		: UINT 	:= AMSPORT_R0_NC; (* used with all axis coupling commands - 12.7.2006 KSt *)  (* 20110511 type changed from INT to UINT *)
	NCNETID_TCMC 				: T_AmsNetId := '';
	NCPORT_TCMC_CAM 			: UINT 	:= AMSPORT_R0_NC; (* 20110511 type changed from INT to UINT *)
	NCPORT_TCMC_CAM_FAST 		: UINT 	:= AMSPORT_R0_NC; (* 20150728 KSt added *)
	NCNETID_TCMC_CAM			: T_AmsNetId := '';
	NCPORT_TCMC_SUPERPOSITION	: UINT 	:= AMSPORT_R0_NCSAF; (* 20140930 KSt added *)
	NCPORT_TCMC_RESET			: UINT 	:= AMSPORT_R0_NC; 	 (* 20211019 KSt added *)
END_VAR
VAR_OUTPUT
	NcDeviceInfoTcMainVersion 	: DWORD;
	NcDeviceInfoTcSubVersion 	: DWORD;
	NcDeviceInfoNcDriverVersion : DWORD;
	NcDeviceInfoNcVersion		: DWORD;
	NcDeviceInfoNcName			: STRING(19);
END_VAR
VAR_OUTPUT CONSTANT	// make visible - KST 24.3.2017
{warning disable C0228}
	Axis 	: _ST_NCADS_Axis;	(* IDXGRP and IDXOFFS constants of axis parameter/status/functions *)
	Table 	: _ST_NCADS_Table;	(* IDXGRP and IDXOFFS constants of table parameter/status/functions *)
{warning restore C0228}
END_VAR
VAR CONSTANT
	NCPORT_TCNCCAMMING_TABLEFUNCTION	: UINT	:=	500;

	(* timeout *)
	tTargetPosTimeOut			: TIME	:= T#6S; (* 20050128 KSt - changed from 5 sec to 6 sec to be later than a NC PEH error (5 sec) *)
	tADSTimeOut   				: TIME	:= T#1S;
	tStopMonitoringTimeOut		: TIME	:= T#100MS;	(* 20111208 KSt - new for stop monitoring (axis in standstill window *)

	NCTOPLC_FEEDBACK_MAXWAITCYCLES : INT := 10; (* maximum number of PLC cycles to wait for a cyclic feedback in NcToPlc after an ADS command *)
END_VAR
VAR
	fbADSRDDEVINFO: ADSRDDEVINFO;
	DeviceVersion: DWORD;
	Init						: BOOL := _F_Init(	DeviceVersion				=>DeviceVersion, 
													NcDeviceInfoTcMainVersion	=>NcDeviceInfoTcMainVersion, 
													NcDeviceInfoTcSubVersion	=>NcDeviceInfoTcSubVersion, 
													NcDeviceInfoNcDriverVersion	=>NcDeviceInfoNcDriverVersion, 
													NcDeviceInfoNcVersion		=>NcDeviceInfoNcVersion, 
													NcDeviceInfoNcName			=>NcDeviceInfoNcName);

END_VAR

;

ACTION ReadDeviceInfo:
(* get current NC version *)
(* this piece of code will be executed just once *)
IF  DeviceVersion = 0 THEN
	IF fbADSRDDEVINFO.ERR THEN
		fbADSRDDEVINFO( RDINFO:= FALSE );
		fbADSRDDEVINFO( RDINFO:= TRUE );
	END_IF

	fbADSRDDEVINFO(
		NETID:= '',
		PORT:= 500,
		RDINFO:= TRUE,
		TMOUT:= T#1s,
		DEVNAME=> NcDeviceInfoNcName,
		DEVVER=> DeviceVersion);

	NcDeviceInfoTcMainVersion := DeviceVersion AND 16#FF;;
	NcDeviceInfoTcSubVersion := (DeviceVersion / 16#100) AND 16#FF;
	NcDeviceInfoNcDriverVersion :=(DeviceVersion / 16#10000) AND 16#FFFF;
	NcDeviceInfoNcVersion := NcDeviceInfoTcMainVersion * 16#1000000 + NcDeviceInfoTcSubVersion * 16#10000 + NcDeviceInfoNcDriverVersion;
END_IF
END_ACTION

END_FUNCTION_BLOCK

// POUs/[Internal]/_F_Init
{attribute 'conditionalshow'}
FUNCTION _F_Init : BOOL
VAR_INPUT
END_VAR
VAR_OUTPUT
	DeviceVersion				: DWORD;
	NcDeviceInfoTcMainVersion 	: DWORD;
	NcDeviceInfoTcSubVersion 	: DWORD;
	NcDeviceInfoNcDriverVersion : DWORD;
	NcDeviceInfoNcVersion		: DWORD;
	NcDeviceInfoNcName			: STRING(19);	
END_VAR
VAR
	_DeviceVersion			: UDINT;
	_DeviceVersionAdr		: PVOID := ADR(_DeviceVersion);
	_DeviceVersionSize		: UDINT := SIZEOF(_DeviceVersion);
	
	hr						: HRESULT;
	//NcVersion				: UDINT;		// hier landet der Wert (BYTE + BYTE + USHORT)
	ipNcCtrl				: ITComObject;
                
	//ErrorId				: UDINT;		// UDINT oder HRESULT?
	ErrorId					: HRESULT;		// eigentlich ist HRESULT richtig
END_VAR

_F_Init := TRUE;
hr := FW_ObjMgr_GetObjectInstance(16#05000000(*OID_TCNC_CTRL*), Tc_GLobal_IID_List.IID_ITComObject, ADR(ipNcCtrl));
IF SUCCEEDED(hr) THEN
	hr := ipNcCtrl.TcGetObjPara(16#0000010A(*PID_AdsVersion*), _DeviceVersionSize, _DeviceVersionAdr, 0);
	ipNcCtrl.TcRelease(); (* immediate release object reference *)
	ipNcCtrl := 0; 
	IF SUCCEEDED(hr) THEN
		(*good case*)
		NcDeviceInfoTcMainVersion := _DeviceVersion AND 16#FF;;
		NcDeviceInfoTcSubVersion := (_DeviceVersion / 16#100) AND 16#FF;
		NcDeviceInfoNcDriverVersion :=(_DeviceVersion / 16#10000) AND 16#FFFF;
		NcDeviceInfoNcVersion := NcDeviceInfoTcMainVersion * 16#1000000 + NcDeviceInfoTcSubVersion * 16#10000 + NcDeviceInfoNcDriverVersion;
		NcDeviceInfoNcName := 'Nc-Server';
		DeviceVersion := _DeviceVersion;
		IF NcDeviceInfoNcVersion >= 16#03011130  (* NC 4400 *) THEN
			TcMCGlobal.NCPORT_TCMC_COUPLING := AMSPORT_R0_NCSAF;
			TcMCGlobal.NCPORT_TCMC_CAM_FAST := AMSPORT_R0_NCSAF;			
		END_IF
	ELSE
		(*bad case, failed getting parameter NC VERSION*)
		ErrorId := hr;
		_F_Init := FALSE;
	END_IF
ELSE
	(*bad case, failed getting object, TcNc driver not loaded or …*)
	ErrorId := hr;
	_F_Init := FALSE;
END_IF

END_FUNCTION

// POUs/[Internal]/_F_GetIndexGroup
{attribute 'conditionalshow'}
FUNCTION _F_GetIndexGroup : _ST_ParaStruct
VAR_INPUT
	ParaNumber	: INT;
	ControlLoopIndex : UINT; // 2016-11-18 KSt
	Mode		: INT; 		(* read/write *)
END_VAR
VAR
	IndexGroup	: UDINT;
	IndexOffset	: UDINT;
	nType 		: _E_ParameterType;
	lrValue		: LREAL;
END_VAR


(* set default values *)
_F_GetIndexGroup.IndexGroup := 0;				(* default *)
_F_GetIndexGroup.IndexOffset:= 0;				(* default *)
_F_GetIndexGroup.ParaType 	:= PARAMETERTYPE_NOTYPE;	(* default *)
_F_GetIndexGroup.LrealSize	:= SIZEOF(lrValue);(* default *)
_F_GetIndexGroup.LrealOffset:= 1;				(* default *)
_F_GetIndexGroup.Port		:= TcMcGlobal.NCPORT_TCMC;	(* default, 2014-07-14 KSt*)
nType						:= PARAMETERTYPE_LREAL;	(* default *)
IndexOffset 				:= 0;				(* default *)
IndexGroup 					:= TcMcGlobal.Axis.Parameter.IDXGRP;	(* default *)

(* check parameter number and determine index group and index offset *)
CASE ParaNumber OF
(*				PLCopen specific parameters *)
(*				Beckhoff specific parameters *)
	AxisId 				:
		IndexOffset := 16#0000_0001;
		nType :=	PARAMETERTYPE_DWORD;
	AxisVeloManSlow :
		IndexOffset := 16#0000_0008;
	AxisVeloManFast :
		IndexOffset := 16#0000_0009;
	AxisVeloMax :
		IndexOffset := 16#0000_0027;
	AxisAcc, MaxAccelerationSystem, MaxAccelerationAppl 	:
		IndexOffset := 16#0000_0101;
	AxisDec, MaxDecelerationSystem, MaxDecelerationAppl 	:
		IndexOffset := 16#0000_0102;
	AxisJerk, MaxJerk, MaxJerkSystem, MaxJerkAppl			:
		IndexOffset := 16#0000_0103;
	AxisMaxVelocity, MaxVelocitySystem, MaxVelocityAppl		:
		IndexOffset := 16#0000_0027;
	AxisRapidTraverseVelocity:
		IndexOffset := 16#0000_000A;
	AxisManualVelocityFast:
		IndexOffset := 16#0000_0009;
	AxisManualVelocitySlow:
		IndexOffset := 16#0000_0008;
	AxisCalibrationVelocityForward:
		IndexOffset := 16#0000_0006;
	AxisCalibrationVelocityBackward:
		IndexOffset := 16#0000_0007;
	AxisJogIncrementForward:
		IndexOffset := 16#0000_0018;
	AxisJogIncrementBackward:
		IndexOffset := 16#0000_0019;
	AxisMinSoftPosLimit, SWLimitNeg:
		IndexOffset := 16#0001_000D;
	AxisMaxSoftPosLimit, SWLimitPos:
		IndexOffset := 16#0001_000E;
	AxisMaxPosLagValue, MaxPositionLag:
		IndexOffset := 16#0002_0012;
	AxisMaxPosLagFilterTime:
		IndexOffset := 16#0002_0013;
	AxisPositionRangeWindow:
		IndexOffset := 16#0000_0010;
	AxisTargetPositionWindow:
		IndexOffset := 16#0000_0016;
	AxisTargetPositionMonitoringTime:
		IndexOffset := 16#0000_0017;
	AxisInTargetTimeout:
		IndexOffset := 16#0000_002A;
	AxisMotionMonitoringWindow:
		IndexOffset := 16#0000_0028;
	AxisMotionMonitoringTime:
		IndexOffset := 16#0000_0012;
	AxisDelayTimeVeloPosition:
		IndexOffset := 16#0000_0104;
	AxisLoopingDistance:
		IndexOffset := 16#0000_0014;
	AxisBacklash:
		IndexOffset := 16#0000_002C;
	AxisRefVeloOnRefOutput:
		IndexOffset := 16#0003_0101;
	AxisOverrideType:
		IndexOffset := 16#0000_0105;
		nType	:=  PARAMETERTYPE_DWORD;
	AxisEnMaxSoftPosLimit, EnableLimitPos:
		IndexOffset := 16#0001_000C;
		nType	:=  PARAMETERTYPE_BOOL;
	AxisEnMinSoftPosLimit, EnableLimitNeg:
		IndexOffset := 16#0001_000B;
		nType	:=  PARAMETERTYPE_BOOL;
	AxisEnPositionLagMonitoring, EnablePosLagMonitoring:
		IndexOffset := 16#0002_0010; (* 4.12.03 KSt, change 0002_0012 to 0002_0010 *)
		nType	:=  PARAMETERTYPE_BOOL;
	AxisEnPositionRangeMonitoring:
		IndexOffset := 16#0000_000F;
		nType	:=  PARAMETERTYPE_BOOL;
	AxisEnTargetPositionMonitoring:
		IndexOffset := 16#0000_0015;
		nType	:=  PARAMETERTYPE_BOOL;
	AxisEnInTargetTimeout:
		IndexOffset := 16#0000_0029;
		nType	:=  PARAMETERTYPE_BOOL;
	AxisEnMotionMonitoring:
		IndexOffset := 16#0000_0011;
		nType	:=  PARAMETERTYPE_BOOL;
	AxisEnLoopingDistance:
		IndexOffset := 16#0000_0013;
		nType	:=  PARAMETERTYPE_BOOL;
	AxisEnBacklashCompensation:
		IndexOffset := 16#0000_002B;
		nType	:=  PARAMETERTYPE_BOOL;
	AxisEnDataPersistence:
		IndexOffset := 16#0000_0030;
		nType	:=  PARAMETERTYPE_BOOL;
	AxisEncoderScalingFactor :
		IndexOffset := 16#0001_0006;
	AxisEncoderScalingNumerator :		(* new since 1/2012 KSt *)
		IndexOffset := 16#0001_0023;
	AxisEncoderScalingDenominator :	(* new since 1/2012 KSt *)
		IndexOffset := 16#0001_0024;
	AxisEncoderOffset :
		IndexOffset := 16#0001_0007;
	AxisEncoderDirectionInverse :
		IndexOffset := 16#0001_0008;
		nType	:=  PARAMETERTYPE_BOOL;
	AxisEncoderMask :
		IndexOffset := 16#0001_0015;
		nType	:=  PARAMETERTYPE_DWORD;
	AxisEncoderMask64 :				(* lword *) (* IndexOffset= 16#0001_0108 *)	(* new since 3/2021 *)
		IndexOffset := 16#0001_0015;
		_F_GetIndexGroup.LrealSize := 0;
		nType	:=  PARAMETERTYPE_LARGE;
	AxisEncoderModuloValue :
		IndexOffset := 16#0001_0009;
	AxisModuloToleranceWindow :
		IndexOffset := 16#0001_001B;
	AxisEnablePosCorrection :
		IndexOffset := 16#0001_0016;
		nType	:=  PARAMETERTYPE_BOOL;
	AxisPosCorrectionFilterTime :
		IndexOffset := 16#0001_0017;
	AxisUnitInterpretation :	(* added 5/20/2008 KSt *)
		IndexOffset := 16#0000_0026;
		nType	:= PARAMETERTYPE_DWORD;
	AxisMotorDirectionInverse :	(* added 1/11/2010 KSt *)
		IndexOffset := 16#0003_0006;
		nType	:=  PARAMETERTYPE_BOOL;
	AxisCycleTime :	(* added 11/29/2010 KSt *)
		IndexOffset := 16#0000_0004;
		nType	:= PARAMETERTYPE_DWORD;
	AxisFastStopSignalType :	(* added 2/5/2011 KSt *)
		IndexOffset := 16#0000_001E;
		nType	:= PARAMETERTYPE_DWORD;
	AxisFastAcc :		(* added 2/5/2011 KSt *)
		IndexOffset := 16#0000_010A;
	AxisFastDec :		(* added 2/5/2011 KSt *)
		IndexOffset := 16#0000_010B;
	AxisFastJerk :		(* added 2/5/2011 KSt *)
		IndexOffset := 16#0000_010C;
		
	(* new since 7/2016 *)
	AxisMaximumAcceleration:		(* lreal *)	(* IndexOffset= 16#0000_00F1 - available in Tc3 *)	(* new since 7/2016 *)
		IndexOffset := 16#0000_00F1;
	AxisMaximumDeceleration:		(* lreal *)	(* IndexOffset= 16#0000_00F2 - available in Tc3 *)	(* new since 7/2016 *)
		IndexOffset := 16#0000_00F2;
	AxisVeloJumpFactor:				(* lreal *)	(* IndexOffset= 16#0000_0106 *)	(* new since 7/2016 *)
		IndexOffset := 16#0000_0106;
	AxisToleranceBallAuxAxis:		(* lreal *)	(* IndexOffset= 16#0000_0108 *)	(* new since 7/2016 *)
		IndexOffset := 16#0000_0108;
	AxisMaxPositionDeviationAuxAxis,(* lreal *)	(* IndexOffset= 16#0000_0109 *) (* new since 5/2018 *)
	AxisMasPositionDeviationAuxAxis:(* lreal *)	(* IndexOffset= 16#0000_0109 *) (* new since 7/2016 *) (* write error MaxPosition, hidden parameter 2018-05-03 KSt *)
		IndexOffset := 16#0000_0109;
	AxisErrorPropagationMode:		(* dword *) (* IndexOffset= 16#0000_001A *)	(* new since 7/2016 *)
		IndexOffset := 16#0000_001A;
		nType	:= PARAMETERTYPE_DWORD;
	AxisErrorPropagationDelay:		(* lreal *)	(* IndexOffset= 16#0000_001B *) (* new since 7/2016 *)
		IndexOffset := 16#0000_001B;
	AxisCoupleSlaveToActualValues:	(* bool *)	(* IndexOffset= 16#0000_001C *)	(* new since 7/2016 *)
		IndexOffset := 16#0000_001C;
		nType	:=  PARAMETERTYPE_BOOL;
	AxisAllowMotionCmdToSlaveAxis:	(* bool *)	(* IndexOffset= 16#0000_0020 *)	(* new since 7/2016 *)
		IndexOffset := 16#0000_0020;
		nType	:=  PARAMETERTYPE_BOOL;
	AxisAllowMotionCmdToExtSetAxis:	(* bool *)	(* IndexOffset= 16#0000_0021 *)	(* new since 7/2016 *)
		IndexOffset := 16#0000_0021;
		nType	:=  PARAMETERTYPE_BOOL;
	AxisEncoderSubMask:				(* dword *) (* IndexOffset= 16#0001_0108 *)	(* new since 7/2016 *)
		IndexOffset := 16#0001_0108;
		nType	:= PARAMETERTYPE_DWORD;
	AxisEncoderSubMask64:			(* lword *) (* IndexOffset= 16#0001_0108 *)	(* new since 3/2021 *)
		IndexOffset := 16#0001_0108;
		_F_GetIndexGroup.LrealSize := 0;
		nType	:= PARAMETERTYPE_LARGE;
	AxisEncoderReferenceSystem:		(* dword *) (* IndexOffset= 16#0001_0019 *)	(* new since 7/2016 *)
		IndexOffset := 16#0001_0019;
		nType	:= PARAMETERTYPE_DWORD;
	AxisEncoderPositionFilterPT1:	(* lreal *)	(* IndexOffset= 16#0001_0010 *)	(* new since 7/2016 *)
		IndexOffset := 16#0001_0010;
	AxisEncoderVelocityFilterPT1:	(* lreal *)	(* IndexOffset= 16#0001_0011 *)	(* new since 7/2016 *)
		IndexOffset := 16#0001_0011;
	AxisEncoderAccelerationFilterPT1:(* lreal *)(* IndexOffset= 16#0001_0012 *)	(* new since 7/2016 *)
		IndexOffset := 16#0001_0012;
	AxisEncoderMode:				(* dword *) (* IndexOffset= 16#0001_000A *)	(* new since 7/2016 *)
		IndexOffset := 16#0001_000A;
		nType	:= PARAMETERTYPE_DWORD;
	AxisEncoderHomingInvDirCamSearch:(* bool *) (* IndexOffset= 16#0001_0101 *)	(* new since 7/2016 *)
		IndexOffset := 16#0001_0101;
		nType	:=  PARAMETERTYPE_BOOL;
	AxisEncoderHomingInvDirSyncSearch:(* bool *)(* IndexOffset= 16#0001_0102 *)	(* new since 7/2016 *)
		IndexOffset := 16#0001_0102;
		nType	:=  PARAMETERTYPE_BOOL;
	AxisEncoderHomingCalibValue:	(* lreal *) (* IndexOffset= 16#0001_0103*)	(* new since 7/2016 *)
		IndexOffset := 16#0001_0103;
	AxisEncoderReferenceMode:		(* dword *) (* IndexOffset= 16#0001_0107 *)	(* new since 7/2016 *)	
		IndexOffset := 16#0001_0107;
		nType	:= PARAMETERTYPE_DWORD;
	AxisRefVeloOutputRatio:			(* lreal *) (* IndexOffset= 16#0003_0102 *)	(* new since 7/2016 *)
		IndexOffset := 16#0003_0102;
	AxisDrivePositionOutputScaling:	(* lreal *) (* IndexOffset= 16#0003_0109 *)	(* new since 7/2016 *)
		IndexOffset := 16#0003_0109;
	AxisDriveVelocityOutputScaling:	(* lreal *) (* IndexOffset= 16#0003_0105 *)	(* new since 7/2016 *)
		(* 2020-05-12 fixed wrong IndexOffset *)
		(* IndexOffset := 16#0003_0000; *)
		IndexOffset := 16#0003_0105;
	AxisDriveVelocityOutputDelay:	(* lreal *) (* IndexOffset= 16#0003_010D *)	(* new since 7/2016 *)
		(* 2020-05-12 fixed wrong IndexOffset *)
		(* IndexOffset := 16#0003_0105; *)
		IndexOffset := 16#0003_010D;
	AxisDriveMinOutputLimitation:	(* lreal *) (* IndexOffset= 16#0003_000B *)	(* new since 7/2016 *)
		IndexOffset := 16#0003_000B;
	AxisDriveMaxOutputLimitation:	(* lreal *) (* IndexOffset= 16#0003_000C *)	(* new since 7/2016 *)
		IndexOffset := 16#0003_000C;
	AxisTorqueInputScaling:			(* lreal *) (* IndexOffset= 16#0003_0031 - available in Tc3 *)	(* new since 7/2016 *)
		IndexOffset := 16#0003_0031;
	AxisTorqueInputFilterPT1:		(* lreal *) (* IndexOffset= 16#0003_0032 - available in Tc3 *)	(* new since 7/2016 *)
		IndexOffset := 16#0003_0032;
	AxisTorqueDerivationInputFilterPT1:	(* lreal *) (* IndexOffset= 16#0003_0033 - available in Tc3 *)	(* new since 7/2016 *)
		IndexOffset := 16#0003_0033;
	AxisTorqueOutputScaling:		(* lreal *) (* IndexOffset= 16#0003_010B *)	(* new since 7/2016 *)
		IndexOffset := 16#0003_010B;
	AxisTorqueOutputDelay:			(* lreal *) (* IndexOffset= 16#0003_010F *)	(* new since 7/2016 *)
		IndexOffset := 16#0003_010F;
	AxisAccelerationOutputScaling:	(* lreal *) (* IndexOffset= 16#0003_010A *)	(* new since 7/2016 *)
		IndexOffset := 16#0003_010A;
	AxisAccelerationOutputDelay:	(* lreal *) (* IndexOffset= 16#0003_010E *)	(* new since 7/2016 *)
		IndexOffset := 16#0003_010E;
	AxisDrivePosOutputSmoothFilterType: (* dword *) (* IndexOffset= 16#0003_0110 *)	(* new since 7/2016 *)
		IndexOffset := 16#0003_0110;
		nType	:= PARAMETERTYPE_DWORD;
	AxisDrivePosOutputSmoothFilterTime:	(* lreal *) (* IndexOffset= 16#0003_0111 *)	(* new since 7/2016 *)
		IndexOffset := 16#0003_0111;
	AxisDrivePosOutputSmoothFilterOrder:(* dword *) (* IndexOffset= 16#0003_0112 *)	(* new since 7/2016 *)
		IndexOffset := 16#0003_0112;
		nType	:= PARAMETERTYPE_DWORD;
	AxisDriveMode:					(* dword *) (* IndexOffset= 16#0003_000A *)	(* new since 7/2016 *)
		IndexOffset := 16#0003_000A;
		nType	:= PARAMETERTYPE_DWORD;
	AxisDriftCompensationOffset:	(* lreal *) (* IndexOffset= 16#0003_0104 *)	(* new since 7/2016 *)
		IndexOffset := 16#0003_0104;
	AxisPositionControlKv:			(* lreal *) (* IndexOffset= 16#0002_0102 *)	(* new since 7/2016 *)
		IndexOffset := 16#0002_0102;
	AxisCtrlVelocityPreCtrlWeight:	(* lreal *) (* IndexOffset= 16#0002_000B *)	(* new since 7/2016 *)
		IndexOffset := 16#0002_000B;
	AxisControllerMode:				(* dword *) (* IndexOffset= 16#0002_000A *)	(* new since 7/2016 *)
		IndexOffset := 16#0002_000A;
		nType	:= PARAMETERTYPE_DWORD;
	AxisCtrlAutoOffset:				(* bool  *) (* IndexOffset= 16#0002_0110 *)	(* new since 7/2016 *)
		IndexOffset := 16#0002_0110;
		nType	:=  PARAMETERTYPE_BOOL;
	AxisCtrlAutoOffsetTimer:		(* lreal *) (* IndexOffset= 16#0002_0115 *)	(* new since 7/2016 *)
		IndexOffset := 16#0002_0115;
	AxisCtrlAutoOffsetLimit:		(* lreal *) (* IndexOffset= 16#0002_0114 *)	(* new since 7/2016 *)
		IndexOffset := 16#0002_0114;
	AxisSlaveCouplingControlKcp:	(* lreal *) (* IndexOffset= 16#0002_010F *)	(* new since 7/2016 *)
		IndexOffset := 16#0002_010F;
	AxisCtrlOutputLimit:			(* lreal *) (* IndexOffset= 16#0002_0100 *)	(* new since 7/2016 *)
		IndexOffset := 16#0002_0100;
		
	(* new since 6/2018 *)
	AxisFadingAccleration:			(* lreal *)	(* IndexOffset= 16#0000_001D *)	(* new since 6/2018 *)
		IndexOffset := 16#0000_001D;

	(* new since 6/2018 *)
	AxisUserDataIdxOffs:			(* udint *)	(* IndexOffset= 16#0000_001D *)	(* new since 6/2018 *)
		IndexOffset := 16#0000_010D;
		nType	:= PARAMETERTYPE_DWORD;

	(* check for status information *)
	AxisTargetPosition:
		IndexGroup := TcMcGlobal.Axis.State.IDXGRP;
		IndexOffset := 16#0000_0013;
	AxisRemainingTimeToGo:
		IndexGroup := TcMcGlobal.Axis.State.IDXGRP;
		IndexOffset := 16#0000_0014;
		_F_GetIndexGroup.LrealSize := 2 * SIZEOF(lrValue);	(* read data structure with two lreal values *)
		_F_GetIndexGroup.LrealOffset := 1;	(* get first lreal value *)
		_F_GetIndexGroup.Port := AMSPORT_R0_NCSAF;		(*  2014-07-14 KSt*)
	AxisRemainingDistanceToGo:
		IndexGroup := TcMcGlobal.Axis.State.IDXGRP;
		IndexOffset := 16#0000_0014;
		_F_GetIndexGroup.LrealSize := 2 * SIZEOF(lrValue);	(* read data structure with two lreal values *)
		_F_GetIndexGroup.LrealOffset := 2;	(* get second lreal value *)
		_F_GetIndexGroup.Port := AMSPORT_R0_NCSAF;		(*  2014-07-14 KSt*)

	(* check for axis function information *)
	AxisGearRatio:
		(* gear ratio is status information in read mode but a function call in write mode *)
		IndexGroup := SEL( Mode=READWRITEPARAMETERMODE_WRITE, TcMcGlobal.Axis.State.IDXGRP, TcMcGlobal.Axis.Functions.IDXGRP );
		IndexOffset := SEL(Mode=READWRITEPARAMETERMODE_WRITE, 16#0000_0022, 16#0000_0042 );
		_F_GetIndexGroup.LrealSize := 4 * SIZEOF(lrValue);	(* read data structure with four lreal values *)
		_F_GetIndexGroup.LrealOffset := 1;	(* get first lreal value *)

	(* system parameters *)
	NcSafCycleTime :
		IndexGroup := 16#1000;
		IndexOffset := 16#0000_0010;
		nType	:= PARAMETERTYPE_DWORD;

	NcSvbCycleTime :
		IndexGroup := 16#1000;
		IndexOffset := 16#0000_0012;
		nType	:= PARAMETERTYPE_DWORD;
ELSE
	nType		:=  PARAMETERTYPE_NOTYPE;	(* not found *)
END_CASE;

IF IndexOffset <> 0 THEN
	IF ControlLoopIndex > 0 AND ControlLoopIndex <= 9 THEN // valid control loop index?
		IF (IndexOffset AND 16#0003_0000) <> 0 THEN // no axis parameter but probably an encoder, drive or controller parameter - 2016-11-18 KSt 
			IndexOffset := IndexOffset + ControlLoopIndex * 16#00100000; //  add control loop index to the index offset 2016-11-18 KSt
		END_IF		
	END_IF
	_F_GetIndexGroup.IndexGroup := IndexGroup;
	_F_GetIndexGroup.IndexOffset := IndexOffset;
	_F_GetIndexGroup.ParaType := nType;
END_IF

END_FUNCTION

// POUs/[Internal]/_F_GetTcDriveObjectId
{attribute 'conditionalshow'}
FUNCTION _F_GetTcDriveObjectId : OTCID
VAR_INPUT
	DriveId			: UDINT;
END_VAR
VAR
END_VAR

IF DriveId <= 0 OR DriveId >= 4096 THEN
	_F_GetTcDriveObjectId := 0;	
ELSE
	_F_GetTcDriveObjectId := 16#05030000 + 16#10 * DriveId;
END_IF

END_FUNCTION

// POUs/[Internal]/_F_GetTcEncoderObjectId
{attribute 'conditionalshow'}
FUNCTION _F_GetTcEncoderObjectId : OTCID
VAR_INPUT
	EncoderId			: UDINT;
END_VAR
VAR
END_VAR

IF EncoderId <= 0 OR EncoderId >= 4096 THEN
	_F_GetTcEncoderObjectId := 0;
ELSE
	_F_GetTcEncoderObjectId := 16#05020000 + 16#10 * EncoderId;
END_IF

END_FUNCTION

// POUs/[Internal]/_F_TcMC_DWORD_TO_HEXSTR2
{attribute 'conditionalshow'}
(*	The iPrecision specifies the minimum number of digits to be printed.
	If the number of digits in the argument is less than iPrecision, the output value is padded on the left with zeros. 
	The value is not truncated when the number of digits exceeds precision.
	If iPrecision is specified as 0 and the in value to be converted is 0, the result is empty string. *)
FUNCTION _F_TcMC_DWORD_TO_HEXSTR2 : T_MaxString
VAR_INPUT
	in				: DWORD;(* DWORD input value *)
	iPrecision		: INT;(* Precision. Number of digits to be printed. *)
	bLoCase			: BOOL := FALSE;  (*Default: use "ABCDEF", if TRUE use "abcdef" characters. *)
END_VAR
VAR
	_FORMAT_HEXASC_CODES							 : ARRAY[0..1, 0..15] OF BYTE 		:=[
	(*lower case*)16#30,16#31,16#32,16#33,16#34,16#35,16#36,16#37,16#38,16#39,16#61,16#62,16#63,16#64,16#65,16#66,
	(*upper case*)16#30,16#31,16#32,16#33,16#34,16#35,16#36,16#37,16#38,16#39,16#41,16#42,16#43,16#44,16#45,16#46];(* Lower and upper case ASCII codes of hexadecimal digits *)

	hex				: ARRAY[0..8] OF BYTE;(* array of ASCII characters (inclusive null delimiter) *)
	iSig			: INT;(* number of significant nibbles *)
	iPad			: INT;(* number of padding zeros *)
	i				: INT;
END_VAR

IF in=0 AND iPrecision = 0 THEN
	_F_TcMC_DWORD_TO_HEXSTR2 := '';
	RETURN;
END_IF
(* Convert nibbles to array of ASCII characters *)
FOR i:= 7 TO 0 BY-1 DO
	hex[ iSig ] := _FORMAT_HEXASC_CODES[SEL(bLoCase,1,0), DWORD_TO_BYTE( SHR( in, i*4 ) AND 16#0F )];
	iSig := SEL( hex[0] = 16#30(* "0" (Null) *), iSig + 1, iSig );
END_FOR
iSig := SEL( iSig = 0, iSig, 1 );

iPad := SEL( iPrecision > iSig, 0, iPrecision - iSig );(* Calculate the number of padding zero characters  *)
iPad := MIN( UDINT_TO_INT(SIZEOF(_F_TcMC_DWORD_TO_HEXSTR2)) - iSig - INT#1, iPad );
MEMSET( ADR( _F_TcMC_DWORD_TO_HEXSTR2 ), 16#30, INT_TO_UDINT(iPad) );(**)
MEMCPY( ADR( _F_TcMC_DWORD_TO_HEXSTR2 ) + iPad, ADR( hex ), INT_TO_UDINT(iSig + 1) );

END_FUNCTION

// POUs/[Internal]/_F_TcMC_IsValidRef
{attribute 'conditionalshow'}
FUNCTION _F_TcMC_IsValidRef : BOOL
VAR_INPUT
	ptr :  PVOID;
	size : UDINT;
END_VAR
VAR
	TcMemoryArea : E_TcMemoryArea; 
END_VAR

IF ptr <> 0 THEN // AXIS REFERENCE CHECK - 2020-09-17 KSt
	TcMemoryArea := F_CheckMemoryArea(ptr, size);
	CASE TcMemoryArea OF 
		1 : _F_TcMC_IsValidRef := TRUE;	// static PLC memory
		2 : _F_TcMC_IsValidRef := TRUE;	// dynamic memory
		ELSE
			_F_TcMC_IsValidRef := FALSE;	// invalid
	END_CASE
ELSE
	_F_TcMC_IsValidRef := FALSE;	// invalid
END_IF

END_FUNCTION

// POUs/[Internal]/_FB_PhasingGeneric
{attribute 'conditionalshow'}
FUNCTION_BLOCK _FB_PhasingGeneric
VAR_IN_OUT
	Master 			: 	AXIS_REF; (*Reference to an axis*)
	Slave 			: 	AXIS_REF; (*Reference to an axis*)
END_VAR
VAR_INPUT
	Execute			:	BOOL;	(* B *)	(* Start the motion at rising edge *)
(*	StartType		: 	UDINT;*)			(* command type start, stop etc, *)
	ContinuousUpdate:	BOOL; (* changes for PhaseShift, Velocity, Acceleration, Deceleration and Jekr can be updated while command is executing *)
	StartType		: 	_E_TcNC_StartPosType;	(* command type start, stop etc, *) (* 20110511 KSt type adaption for TC3 *)
	PhaseShift		:	LREAL;	(* B *)	(* Target position for the motion *)
	PhasingType		: 	E_PhasingType;	(* type of phase shift value, absolute or relative *)
	Velocity			:	LREAL;	(* E *)	(* Value of the maximum velocity *)
	Acceleration		:	LREAL;	(* E *)	(* Value of the maximum acceleration *)
	Deceleration		:	LREAL;	(* E *)	(* Value of the maximum deceleration *)
	Jerk				:	LREAL;	(* E *)	(* Value of the maximum jerk *)
	BufferMode		:	MC_BufferMode;		(* E *)
	Options			: 	ST_PhasingOptions;	(* V *)	(* optional parameters *)
END_VAR
VAR_OUTPUT
	Done			:	BOOL;	(* B *)
	Busy			: 	BOOL;	(* E *)
	Active			: 	BOOL;	(* E *)
	CommandAborted	:	BOOL;	(* E *)
	Error			:	BOOL;	(* B *)
{attribute 'displaymode':='hex'}
	ErrorID			:	UDINT;	(* E *)
	PhaseShiftFeedback : 	LREAL;	(* E *)
END_VAR
VAR
	LastExecutionResult: 	_ST_FunctionBlockResults;
	ADSbusy		: 	BOOL;
	iState			:	_E_TcMC_STATES := STATE_INITIALIZATION;
(*	fbAdsReadWrite	: 	ADSRDWRTEX;*)
	fbAdsWrite		: 	ADSWRITE;
	sNcPhasing		: 	_ST_TcNC_PhasingRequest;
	PhasingStarted: BOOL;
	iContinuousUpdate: BOOL;
END_VAR
VAR
{attribute 'hide'}
	fbTrigger			:	R_TRIG;
{attribute 'hide'}
	fbTimeOut		: 	TON;
{attribute 'hide'}
	pPhasingState: POINTER TO _E_PhasingState;
END_VAR

(* ====================================================================== *)
(* *)
(* ====================================================================== *)
fbTrigger(CLK:= Execute);

CASE iState OF
STATE_INITIALIZATION:	(* *)
	Busy := FALSE;
	Active := FALSE;

	IF NOT Execute THEN
		Done := FALSE;
		CommandAborted := FALSE;
		Error := FALSE;			(* reset at falling edge of Execute *)
		ErrorID := 0;
	END_IF;

   	IF fbTrigger.Q THEN
		(* initialize output values *)
		Done := FALSE;
		Busy := TRUE;
		CommandAborted := FALSE;
		Error := FALSE;
		ErrorID := 0;
		LastExecutionResult.Done := FALSE;
		LastExecutionResult.CommandAborted := FALSE;
		LastExecutionResult.Error := FALSE;
		LastExecutionResult.ErrorID := 0;
		PhaseShiftFeedback := 0;
		fbTimeOut(IN:= FALSE);
		fbAdsWrite(WRITE:=FALSE);

		(* fill structure *)
		sNcPhasing.nPhasingType	:= PhasingType;
		sNcPhasing.nControlMask 	:= 0;
		sNcPhasing.fPhaseShift	:= PhaseShift;
		sNcPhasing.fVelo			:= Velocity;
		sNcPhasing.fAcc			:= Acceleration;
		sNcPhasing.fDec			:= Deceleration;
		sNcPhasing.fJerk			:= Jerk;
		sNcPhasing.nMasterAxisID	:= Master.NcToPlc.AxisId;
		sNcPhasing.nBufferMode	:= BufferMode;	(* not yet implemented *)
		sNcPhasing.fBlendingPos	:= 0;				(* not yet implemented *)
		
		iContinuousUpdate := ContinuousUpdate;

		fbAdsWrite.PORT := SEL(Slave.ADS.Port = 0, Slave.ADS.port, AMSPORT_R0_NCSAF);	(* KSt, 20090123 *)
		fbAdsWrite(	NETID:= TcMcGlobal.NCNETID_TCMC,
					IDXGRP:= TcMcGlobal.Axis.Functions.IDXGRP+Slave.NcToPlc.AxisId,
					IDXOFFS:= TcMcGlobal.Axis.Functions.IDXOFFS.PHASINGREQEUST,
					LEN:= SIZEOF(sNcPhasing),
					SRCADDR:= ADR(sNcPhasing),
					WRITE:= TRUE,
					TMOUT:= TcMcGlobal.tADSTimeOut );

		iState := STATE_ORDER;
	END_IF;

STATE_ORDER:  (* wait until command is accepted *)
	fbAdsWrite(WRITE:= TRUE);
	IF NOT fbAdsWrite.Busy THEN
		IF fbAdsWrite.Err THEN
			Error := TRUE;
			ErrorID := fbAdsWrite.ErrId;
			iState := STATE_INITIALIZATION;
		ELSE
			PhaseShiftFeedback := sNcPhasing.fPhaseShift;
			Active := TRUE;
			PhasingStarted := F_AxisPhasingActive(Slave.NcToPlc.StateDWord) ;
			pPhasingState := ADR(Slave._internal.PhasingState); // KSt 20190703 store phasing state globaly
			pPhasingState^ := SEL(PhasingType=NC_PHASINGTYPE_STOP, PhasingActivated, PhasingAborted ); // KSt 20190703 store phasing state globaly
			iState := STATE_RUNNING;
		END_IF;
	END_IF;

STATE_RUNNING:  (* wait until axis stands still *)
	IF F_AxisPhasingActive(Slave.NcToPlc.StateDWord) THEN 	(* KSt, 29.4.2008 *)
		PhasingStarted := TRUE;
	ELSIF PhasingStarted OR (StartType=TCNC_START_STOPANDLOCK) (* AND phasing  finished now *) THEN
		// Done := TRUE; // KSt 20190703
		CommandAborted := SEL(Slave._internal.PhasingState=PhasingAborted AND (StartType<>TCNC_START_STOPANDLOCK), FALSE, TRUE ); // KSt 20190703 Done or CommandAborted depending on phasing state 
		Done := NOT CommandAborted; // KSt 20190703 Done or CommandAborted depending on phasing state 
		pPhasingState := ADR(Slave._internal.PhasingState); // KSt 20190703 store phasing state globaly
		pPhasingState^ := PhasingInactive; 					// KSt 20190703 store phasing state globaly
		iState := STATE_INITIALIZATION;
	ELSE (* phasing operation did not start so far *)
		(* check for superposition not beeing started (KSt, 12.01.2004) *)
		fbTimeOut(IN:= TRUE, PT:= T#50ms);
		IF fbTimeOut.Q THEN
			(*	when the ADS command comes back without any error but
				the phasing operation does not start anyway, we assume that  
				a very short phasing operation has already been executed. 
			*)
			Done := TRUE; (* after short timeout *)
			iState := STATE_INITIALIZATION;
		END_IF;
	END_IF

	IF iContinuousUpdate AND NOT ContinuousUpdate THEN
		iContinuousUpdate := FALSE;
	END_IF
	
	IF iContinuousUpdate AND iState <> STATE_INITIALIZATION THEN
		IF (sNcPhasing.fPhaseShift	<> PhaseShift)
		  OR (sNcPhasing.fVelo		<> Velocity)
		  OR (sNcPhasing.fAcc		<> Acceleration)
		  OR (sNcPhasing.fDec		<> Deceleration)
		  OR (sNcPhasing.fJerk		<> Jerk)
		THEN
			sNcPhasing.nControlMask.0 	:= TRUE;
			sNcPhasing.fPhaseShift	:= PhaseShift;
			sNcPhasing.fVelo		:= Velocity;
			sNcPhasing.fAcc			:= Acceleration;
			sNcPhasing.fDec			:= Deceleration;
			sNcPhasing.fJerk		:= Jerk;
			
			fbAdsWrite(WRITE:=FALSE);
			fbAdsWrite(WRITE:=TRUE);

			iState := STATE_ORDER;
		END_IF
	END_IF
	
ELSE  (* CASE : Unknown program state *)
	Error := TRUE;
	ErrorID := 16#FFFFFFFF;
	iState:= STATE_INITIALIZATION;
END_CASE

ADSbusy := fbAdsWrite.BUSY;
IF iState=STATE_INITIALIZATION THEN
	(* reset Busy immediately  when sequence ends *)
	IF Busy THEN
		LastExecutionResult.Done := Done;
		LastExecutionResult.CommandAborted := CommandAborted;
		LastExecutionResult.Error := Error;
		LastExecutionResult.ErrorID := ErrorID;
	END_IF
	Busy := FALSE;
	Active := FALSE;
END_IF

END_FUNCTION_BLOCK

// POUs/[Internal]/_FB_ReadWriteParameter
{attribute 'conditionalshow'}
FUNCTION_BLOCK _FB_ReadWriteParameter
VAR_IN_OUT
	Axis				:	AXIS_REF; (*Reference to an axis*)
END_VAR
VAR_INPUT
	Enable			:	BOOL;
	ParameterNumber	:	MC_AxisParameter;
	Mode			:	INT; 		(* read/write *)
//	ParameterType	:	INT;		(* bool/ not  bool *)	(* removed 2018-11-22 KSt - not required *)
	ParameterPointer: 	PVOID;	// for structured parameters - KSt 2021-03-04
	ParameterSize	:	USINT; 	// for structured parameters  - KSt 2021-03-04
END_VAR
VAR_OUTPUT
	Done			:	BOOL;
	Busy: BOOL;
	Error			:	BOOL;
{attribute 'displaymode':='hex'}
	ErrorID			:	UDINT;
	ADSbusy: BOOL;
END_VAR
VAR_IN_OUT
	ValueLreal		:	LREAL;
	ValueDword		:	DWORD;
	ValueBool		:	BOOL;
END_VAR
VAR
	iState			:	_E_TcMC_STATES := STATE_INITIALIZATION;
	fbAdsRead		:	ADSREAD;
	fbAdsWrite		:	ADSWRITE;

	dwValue			:	DWORD;
	lrValue			:	ARRAY[1..10] OF LREAL;
	NcBoolValue		:	UINT;

	bStarted		:	BOOL;
	stParaStruct	:	_ST_ParaStruct;
	n: INT;
	i: INT;
END_VAR
VAR CONSTANT
(*	ParaDWORD		:	INT:= 1;*)
	ParaLREAL		:	INT := 2;
(*	ParaBOOL		:	INT := 3;*)
END_VAR

IF NOT _F_TcMC_IsValidAxisRef(Axis) THEN // AXIS REFERENCE CHECK - 2020-09-17 KSt
	Error := TRUE;
	ErrorID := MC_ERROR_INVALIDREFERENCE;
	RETURN;
END_IF

(* ====================================================================== *)
(* *)
(* ====================================================================== *)

CASE iState OF
STATE_INITIALIZATION:	(* Ruhezustand *)
	Busy := FALSE;
    	IF Enable THEN
		(* initialize output values *)
		Done := FALSE;
		Error := FALSE;
		ErrorID := 0;

		stParaStruct.LrealSize := SIZEOF(lrValue[1]);
		stParaStruct.LrealOffset := 1;
		stParaStruct.Port := TcMcGlobal.NCPORT_TCMC; (* 2014-07-14 KSt *)

		(* some parameters are read immediately out of the cyclic axis interfaces *)
		(* other parameters are read via ADS, F_GetIndexGroup finds the required ADS parameters in this case *)
		IF Mode=READWRITEPARAMETERMODE_READ THEN
			CASE ParameterNumber OF
				CommandedPosition :
					stParaStruct.IndexOffset := 16#0000_0000;
					stParaStruct.IndexGroup := 0;
					stParaStruct.ParaType := ParaLreal;
					ValueLreal := Axis.NcToPlc.SetPos;
					Done := TRUE;
				ActualVelocity:
					stParaStruct.IndexOffset := 16#0000_0000;
					stParaStruct.IndexGroup := 0;
					stParaStruct.ParaType := ParaLreal;
					ValueLreal := Axis.NcToPlc.ActVelo;
					Done := TRUE;
				CommandedVelocity:
					stParaStruct.IndexOffset := 16#0000_0000;
					stParaStruct.IndexGroup := 0;
					stParaStruct.ParaType := ParaLreal;
					ValueLreal := Axis.NcToPlc.SetVelo;
					Done := TRUE;
				ELSE
					(* check index offset *)
					stParaStruct := _F_GetIndexGroup(ParaNumber := ParameterNumber, ControlLoopIndex := Axis.NcToPlc.ControlLoopIndex, Mode:=Mode);
			END_CASE;
		ELSE
			(* check index offset *)
			stParaStruct := _F_GetIndexGroup(ParaNumber := ParameterNumber, ControlLoopIndex := Axis.NcToPlc.ControlLoopIndex, Mode:=Mode);
		END_IF
		IF NOT Done THEN
			IF stParaStruct.ParaType = PARAMETERTYPE_LARGE AND (ParameterPointer=0 OR ParameterSize=0) THEN
				Error:=TRUE;
				ErrorID := MC_ERROR_COMMAND_NOT_ALLOWED; // LARGE > LREAL parameter can only be read with MC_ReadLargeParameter - 20210412 KSt
			ELSIF stParaStruct.ParaType <> PARAMETERTYPE_LARGE AND (ParameterPointer<>0 OR ParameterSize<>0) THEN
				Error:=TRUE;
				ErrorID := MC_ERROR_COMMAND_NOT_ALLOWED; // other parameter cannot be read with MC_ReadLargeParameter - 20210412 KSt
			ELSE
				Busy := TRUE;
				iState := STATE_ORDER;
			END_IF
		END_IF
	ELSE
		Done := FALSE; (* reset with Enable=FALSE *)
		Error := FALSE;			(* reset at falling edge of Execute *)
		ErrorID := 0;
	END_IF
END_CASE

CASE iState OF
STATE_INITIALIZATION:
	;	(* already done before *)
STATE_ORDER :
		(* read via ADS *)
// removed 2018-11-22 KSt - not required (has not been used) 
//		IF FALSE AND (stParaStruct.ParaType <> ParameterType) (* no check !!*)
//		THEN
//			(* type mismatch *)
//			Done := FALSE;
//			ErrorID := MC_ERROR_COMMAND_NOT_ALLOWED;
//			Error := TRUE;
//		ELSIF stParaStruct.ParaType <> PARAMETERTYPE_NOTYPE THEN

		IF stParaStruct.ParaType <> PARAMETERTYPE_NOTYPE THEN
			CASE Mode OF
(*------------------ Read parameter ---------------------------------------------------------------*)
				READWRITEPARAMETERMODE_READ	:
					IF stParaStruct.IndexGroup = 16#1000 (* no axis parameter *) AND
						(stParaStruct.IndexOffset=16#10 OR stParaStruct.IndexOffset=16#12) (* NC SAF or SVB cycle time *)
						THEN
						IF stParaStruct.ParaType=PARAMETERTYPE_DWORD THEN	(* read DWORD *)
								fbAdsRead(	NETID:= TcMcGlobal.NCNETID_TCMC,
(*									PORT:= TcMcGlobal.NCPORT_TCMC,*) (* 2014-07-14 KSt *)
									PORT:= stParaStruct.Port, (* 2014-07-14 KSt *)
									IDXGRP:= stParaStruct.IndexGroup,
									IDXOFFS:= stParaStruct.IndexOffset,
									LEN:= SIZEOF(dwValue),
									DESTADDR:= ADR(dwValue),
									READ:= TRUE,
									TMOUT:= TcMcGlobal.tADSTimeOut);
									ValueDword := 0;
									ValueLreal := DWORD_TO_LREAL(dwValue) * LREAL#100.0E-9;	(* convert to time value (SAF or SVB cycle time)*)
									ValueBool := 0;
						ELSE
							ErrorID := MC_ERROR_COMMAND_NOT_ALLOWED;
							Error := TRUE;
						END_IF

					ELSE (* axis data *)
						CASE stParaStruct.ParaType OF
							PARAMETERTYPE_DWORD :	(* read DWORD *)
								fbAdsRead(	NETID:= TcMcGlobal.NCNETID_TCMC,
(*									PORT:= TcMcGlobal.NCPORT_TCMC,*) (* 2014-07-14 KSt *)
									PORT:= stParaStruct.Port, (* 2014-07-14 KSt *)
									IDXGRP:= stParaStruct.IndexGroup+Axis.NcToPlc.AxisId,
									IDXOFFS:= stParaStruct.IndexOffset,
									LEN:= SIZEOF(dwValue),
									DESTADDR:= ADR(dwValue),
									READ:= TRUE,
									TMOUT:= TcMcGlobal.tADSTimeOut);
									ValueDword := dwValue; (* 20110511 KSt type conversion deleted for Tc3 *)
									ValueLreal := DWORD_TO_LREAL (dwValue);
									ValueBool := DWORD_TO_BOOL(dwValue);
								IF stParaStruct.IndexOffset=16#0000_0004 THEN
									ValueDword := 0;
									ValueLreal := DWORD_TO_LREAL(dwValue) * LREAL#1.0E-6;	(* convert to time value (axis cycle time)*)
									ValueBool := 0;
								END_IF
							PARAMETERTYPE_LREAL :		(* read LREAL *)
								fbAdsRead(	NETID:= TcMcGlobal.NCNETID_TCMC,
(*									PORT:= TcMcGlobal.NCPORT_TCMC,*) (* 2014-07-14 KSt *)
									PORT:= stParaStruct.Port, (* 2014-07-14 KSt *)
									IDXGRP:= stParaStruct.IndexGroup+Axis.NcToPlc.AxisId,
									IDXOFFS:= stParaStruct.IndexOffset,
									LEN:= MIN(SIZEOF(lrValue), stParaStruct.LrealSize),
									DESTADDR:= ADR(lrValue),
									READ:= TRUE,
									TMOUT:=  TcMcGlobal.tADSTimeOut);
									ValueLreal := lrValue[stParaStruct.LrealOffset];
									IF ValueLreal > 16#FFFF_FFFF THEN	(* 31.5.2007 KSt - avoid FPU exception *)
										ValueDword := 0;
										ValueBool := TRUE;
									ELSIF ValueLreal < -16#8000_0000 THEN 	(* 31.5.2007 KSt - avoid FPU exception *)
										ValueDword := 0;
										ValueBool := TRUE;
									ELSE
										ValueDword := LREAL_TO_DWORD(lrValue[stParaStruct.LrealOffset]); 	(* 31.5.2007 KSt - existing code *)
										ValueBool := LREAL_TO_BOOL(lrValue[stParaStruct.LrealOffset]);		(* 31.5.2007 KSt - existing code *)
									END_IF
	
							PARAMETERTYPE_BOOL :		(* read bool *)
								fbAdsRead(	NETID:= TcMcGlobal.NCNETID_TCMC,
(*									PORT:= TcMcGlobal.NCPORT_TCMC,*) (* 2014-07-14 KSt *)
									PORT:= stParaStruct.Port, (* 2014-07-14 KSt *)
									IDXGRP:= stParaStruct.IndexGroup+Axis.NcToPlc.AxisId,
									IDXOFFS:= stParaStruct.IndexOffset,
									LEN:= SIZEOF(NcBoolValue),
									DESTADDR:= ADR(NcBoolValue),
									READ:= TRUE,
									TMOUT:=  TcMcGlobal.tADSTimeOut);
									ValueBool := UINT_TO_BOOL(NcBoolValue);
									ValueDword := UINT_TO_DWORD(NcBoolValue);
									ValueLreal := UINT_TO_LREAL (NcBoolValue);
	
							PARAMETERTYPE_LARGE :		(* read large parameters e. g. struct or LWORD - KSt 2021-03 *)
								fbAdsRead(	NETID:= TcMcGlobal.NCNETID_TCMC,
									PORT:= stParaStruct.Port,
									IDXGRP:= stParaStruct.IndexGroup+Axis.NcToPlc.AxisId,
									IDXOFFS:= stParaStruct.IndexOffset,
									LEN:= ParameterSize,
									DESTADDR:= ParameterPointer,
									READ:= TRUE,
									TMOUT:=  TcMcGlobal.tADSTimeOut);
									ValueLreal := 0;
									ValueDword := 0;
									ValueBool := FALSE;	
						END_CASE;
					END_IF
(*------------------ Write parameter ---------------------------------------------------------------*)
				READWRITEPARAMETERMODE_WRITE	:
					IF stParaStruct.IndexGroup = 16#1000 THEN (* no axis parameter *)
						ErrorID := MC_ERROR_COMMAND_NOT_ALLOWED;
						Error := TRUE;
					ELSE
						CASE stParaStruct.ParaType OF
							PARAMETERTYPE_DWORD:	(* read DWORD *)
								ValueDword := LREAL_TO_DWORD(ValueLreal);
								fbAdsWrite(	NETID:= TcMcGlobal.NCNETID_TCMC,
(*									PORT:= TcMcGlobal.NCPORT_TCMC,*) (* 2014-07-14 KSt *)
									PORT:= stParaStruct.Port, (* 2014-07-14 KSt *)
									IDXGRP:= stParaStruct.IndexGroup+Axis.NcToPlc.AxisId,
									IDXOFFS:= stParaStruct.IndexOffset,
									LEN:= SIZEOF(ValueDword),
									SRCADDR:= ADR(ValueDword),
									WRITE:= TRUE,
									TMOUT:= TcMcGlobal.tADSTimeOut);
	
							PARAMETERTYPE_LREAL :		(* read LREAL *)
								n := SIZEOF(lrValue) / SIZEOF(lrValue[1]);
								FOR i := 1 TO n DO lrValue[i] := 0; END_FOR
								lrValue[stParaStruct.LrealOffset] := ValueLreal;
								fbAdsWrite(	NETID:= TcMcGlobal.NCNETID_TCMC,
(*									PORT:= TcMcGlobal.NCPORT_TCMC,*) (* 2014-07-14 KSt *)
									PORT:= stParaStruct.Port, (* 2014-07-14 KSt *)
									IDXGRP:= stParaStruct.IndexGroup+Axis.NcToPlc.AxisId,
									IDXOFFS:= stParaStruct.IndexOffset,
									LEN:= MIN(SIZEOF(lrValue), stParaStruct.LrealSize),
									SRCADDR:= ADR(lrValue),
									WRITE:= TRUE,
									TMOUT:=  TcMcGlobal.tADSTimeOut);
	
							PARAMETERTYPE_BOOL :		(* read BOOL *)
								NcBoolValue := BOOL_TO_UINT(ValueBool);
								fbAdsWrite(	NETID:= TcMcGlobal.NCNETID_TCMC,
(*									PORT:= TcMcGlobal.NCPORT_TCMC,*) (* 2014-07-14 KSt *)
									PORT:= stParaStruct.Port, (* 2014-07-14 KSt *)
									IDXGRP:= stParaStruct.IndexGroup+Axis.NcToPlc.AxisId,
									IDXOFFS:= stParaStruct.IndexOffset,
									LEN:= SIZEOF(NcBoolValue),
									SRCADDR:= ADR(NcBoolValue),
									WRITE:= TRUE,
									TMOUT:=  TcMcGlobal.tADSTimeOut);

							PARAMETERTYPE_LARGE :		(* read large parameters e. g. struct or LWORD - KSt 2021-03 *)
								fbAdsWrite(	NETID:= TcMcGlobal.NCNETID_TCMC,
									PORT:= stParaStruct.Port, 
									IDXGRP:= stParaStruct.IndexGroup+Axis.NcToPlc.AxisId,
									IDXOFFS:= stParaStruct.IndexOffset,
									LEN:= ParameterSize,
									SRCADDR:= ParameterPointer,
									WRITE:= TRUE,
									TMOUT:=  TcMcGlobal.tADSTimeOut);
						END_CASE;
				END_IF
			END_CASE;

			bStarted := TRUE;
			CASE Mode OF
(*------------------ Read parameter ---------------------------------------------------------------*)
				READWRITEPARAMETERMODE_READ	:
					IF NOT fbAdsRead.Busy THEN
						bStarted := FALSE;
						iState := STATE_RUNNING;
					END_IF;
(*------------------ Write parameter ---------------------------------------------------------------*)
				READWRITEPARAMETERMODE_WRITE	:
					IF NOT fbAdsWrite.BUSY THEN
						bStarted := FALSE;
						iState := STATE_RUNNING;
					END_IF;
			END_CASE;
		ELSE
			Done := FALSE;
			ErrorID := MC_ERROR_COMMAND_NOT_ALLOWED;
			Error := TRUE;
			iState := STATE_INITIALIZATION;
		END_IF;

STATE_RUNNING:  (* wait *)
	IF NOT Error THEN
		CASE Mode OF
		(*------------------ Read parameter ---------------------------------------------------------------*)
			READWRITEPARAMETERMODE_READ	:
				IF fbAdsRead.Err THEN
					ValueLreal := 0.0;
					ValueDword := 0;
					ValueBool := FALSE;
					Done := FALSE;
					ErrorID := fbAdsRead.ErrId;
					Error := TRUE;
					fbAdsRead(READ := FALSE);
					iState := STATE_INITIALIZATION;
				ELSE
					Done := TRUE;
					fbAdsRead(READ := FALSE);
			 		iState:=STATE_INITIALIZATION;
				END_IF;
	(*------------------ Write parameter ---------------------------------------------------------------*)
			READWRITEPARAMETERMODE_WRITE	:
				IF fbAdsWrite.Err THEN
					Done := FALSE;
					ErrorID := fbAdsWrite.ErrId;
					Error := TRUE;
					fbAdsWrite(WRITE := FALSE);
					iState := STATE_INITIALIZATION;
				ELSE
					Done := TRUE;
					fbAdsWrite(WRITE := FALSE);
			 		iState:=STATE_INITIALIZATION;
				END_IF;
		END_CASE;
	ELSE
 		iState:=STATE_INITIALIZATION;
	END_IF;

ELSE  (* CASE : Unknown program state *)
	Error := TRUE;
	ErrorID := 16#FFFFFFFF;
	iState:=STATE_INITIALIZATION;
END_CASE;

ADSbusy := fbAdsWrite.BUSY OR fbAdsRead.BUSY;
IF iState=STATE_INITIALIZATION THEN
	(* reset Busy immediately  when sequence ends *)
	Busy := FALSE;
END_IF

END_FUNCTION_BLOCK

// POUs/Administrative/Status and Parameter/MC_ReadLargeParameter
FUNCTION_BLOCK MC_ReadLargeParameter
(*	This Function Block returns the value of a vendor specific parameter *)
VAR_IN_OUT
	Axis			:	AXIS_REF; (*Reference to an axis*)
END_VAR
VAR_INPUT
	Enable			:	BOOL;		
	ParameterNumber	:	MC_AxisParameter; // 2023-03 KSt changed from INT to MC_AxisParameter		
	ParameterPointer: 	PVOID;	// for structured parameters - KSt 2021-03-04
	ParameterSize	:	USINT; 	// for structured parameters  - KSt 2021-03-04
	ReadMode		:	E_ReadMode := ReadMode_Once;	 (* Beckhoff proprietary input *)
END_VAR
VAR_OUTPUT
	Valid			:	BOOL;		
	Busy			: 	BOOL;		
	Error			:	BOOL;		
{attribute 'displaymode':='hex'}
	ErrorID			:	UDINT;		
//	Value			:	LREAL;		
END_VAR
VAR
	ADSbusy		: 	BOOL;
	fbReadWriteParameter: 	_FB_ReadWriteParameter;
END_VAR
VAR
{attribute 'conditionalshow'}
	lrValue 		: 	LREAL;
{attribute 'conditionalshow'}
	dwValue 		: 	DWORD;
{attribute 'conditionalshow'}
	bValue 			: 	BOOL;
{attribute 'conditionalshow'}
	bStarted		:	BOOL;
{attribute 'conditionalshow'}
	fbTrigger		 	: 	R_TRIG;
END_VAR

(* ====================================================================== *)
(* *)
(* ====================================================================== *)
IF NOT Enable THEN
	Valid := FALSE;
	Error := FALSE;			(* reset at falling edge of Execute - just ErrorID will be kept til next rising edge *)
	ErrorID := 0;
END_IF
IF ReadMode = ReadMode_Once THEN
	fbTrigger(CLK:= Enable);
	IF fbTrigger.Q AND NOT bStarted THEN
		bStarted := TRUE;
		Valid := FALSE;
		Error := FALSE;
		ErrorID := MC_ERROR_NO_ERROR;
	END_IF;
ELSE
	IF Enable AND NOT bStarted THEN
		bStarted := TRUE;
		Valid := FALSE;
		Error := FALSE;
		ErrorID := MC_ERROR_NO_ERROR;
	END_IF;
	IF NOT Enable AND NOT bStarted THEN
		Valid := FALSE;
		Error := FALSE;
		ErrorID := MC_ERROR_NO_ERROR;
	END_IF;
END_IF;

IF bStarted THEN
//	nParatype := PARAMETERTYPE_LARGE;
	fbReadWriteParameter(Enable:= TRUE, ParameterNumber:= ParameterNumber, Mode:= READWRITEPARAMETERMODE_READ,
						(*ParameterType:=nParatype,*) Axis:= Axis, ValueLreal:= lrValue, ValueDword := dwValue, ValueBool := bValue,
						ParameterPointer := ParameterPointer, ParameterSize:=ParameterSize);
	IF fbReadWriteParameter.Done THEN
		bStarted := FALSE;
		Valid := TRUE;
		fbReadWriteParameter(Enable:= FALSE, ParameterNumber:= ParameterNumber, Mode:= READWRITEPARAMETERMODE_READ,
						(*ParameterType:= nParatype,*) Axis:= Axis, ValueLreal:= lrValue, ValueDword := dwValue, ValueBool := bValue);
	END_IF;
	IF fbReadWriteParameter.Error THEN
		bStarted := FALSE;
		Valid := FALSE;
		Error := TRUE;
		ErrorID := fbReadWriteParameter.ErrorID;
		fbReadWriteParameter(Enable:= FALSE, ParameterNumber:= ParameterNumber, Mode:= READWRITEPARAMETERMODE_READ,
						(*ParameterType:= nParatype,*) Axis:= Axis, ValueLreal:= lrValue, ValueDword := dwValue, ValueBool := bValue);
	END_IF;
END_IF;

ADSbusy := fbReadWriteParameter.ADSbusy;
Busy := (Enable AND ReadMode<>ReadMode_Once) OR bStarted;

END_FUNCTION_BLOCK

// POUs/[Internal]/_FB_WriteParameterPersistent
{attribute 'conditionalshow'}
FUNCTION_BLOCK _FB_WriteParameterPersistent
VAR_IN_OUT
	Axis: AXIS_REF; (*Reference to an axis*)
END_VAR
VAR_INPUT
	Execute: BOOL;
	ParameterNumber: MC_AxisParameter; // 2023-03 KSt changed from INT to MC_AxisParameter
	Value: LREAL;
//	ParameterType: INT;	(* removed 2018-11-22 KSt - not required *)
	ParameterPointer: 	PVOID;	// for structured parameters - KSt 2021-03-04
	ParameterSize	:	USINT; 	// for structured parameters  - KSt 2021-03-04
END_VAR
VAR_OUTPUT
	Done: BOOL;
	Busy: BOOL;
	Error: BOOL;
{attribute 'displaymode':='hex'}
	ErrorID: UDINT;
END_VAR
VAR
	ADSbusy: BOOL;
	fbReadWriteParameter: _FB_ReadWriteParameter;
	state: INT;
	stParaStruct: _ST_ParaStruct;
	//	nParatype 		:	_E_ParameterType;
{attribute 'conditionalshow'}
	iParameterNumber: MC_AxisParameter; // 2023-03 KSt changed from INT to MC_AxisParameter
{attribute 'conditionalshow'}
	lrValue: LREAL;
{attribute 'conditionalshow'}
	dwValue: DWORD;
{attribute 'conditionalshow'}
	bValue: BOOL;
	bValueWord: UINT;
{attribute 'conditionalshow'}
	fbTrigger: R_TRIG;
	fbAdsWriteSystemService: ADSWRITE;
	aCmdBuffer: ARRAY[1..256] OF BYTE; // memory for AdsAddInitCommand plus additional strings (maximal size= 8 + 40 + 80 + 1 + 80 + 1 = 210)
	pCmd: POINTER TO AdsAddInitCommand;
	pByte: POINTER TO BYTE;
{attribute 'conditionalshow'}
	sKey: STRING;
{attribute 'conditionalshow'}
	sMsg: STRING;
{attribute 'conditionalshow'}
	sTmp: STRING;
	IG: UDINT;
	IO: UDINT;
	size: UINT;
	valuesize: UINT;
END_VAR

IF NOT _F_TcMC_IsValidAxisRef(Axis) THEN // AXIS REFERENCE CHECK - 2020-09-17 KSt
	Error := TRUE;
	ErrorID := MC_ERROR_INVALIDREFERENCE;
	RETURN;
END_IF

fbTrigger(CLK:= Execute);

CASE state OF
	0 :
	IF NOT Execute THEN
		Done := FALSE;
		Error := FALSE;			(* reset at falling edge of Execute *)
		ErrorID := 0;
	END_IF
	IF fbTrigger.Q THEN
		Busy := TRUE;
		Done := FALSE;
		Error := FALSE;
		ErrorID := MC_ERROR_NO_ERROR;
//		IF ParameterType=PARAMETERTYPE_BOOL THEN
//			bValue := Value<>0;
//			bValueWord := SEL(bValue, 0, 1);
//		END_IF*)
		fbReadWriteParameter(Enable:= FALSE, Axis:=Axis, ValueLreal:= lrValue, ValueDword := dwValue, ValueBool := bValue);
		fbAdsWriteSystemService(WRITE:= FALSE);
		iParameterNumber := ParameterNumber; // save parameter number 
		// convert value to several data types
		lrValue := Value;
		bValue := lrValue<>0; (* 2010-05-04 KST - to write bool parameters with MC_WriteParameter as well *)
		bValueWord := SEL(bValue, 0, 1);
		dwValue := LREAL_TO_DWORD(lrValue);
		fbReadWriteParameter(Enable:= TRUE, ParameterNumber:= iParameterNumber, Mode:= READWRITEPARAMETERMODE_WRITE,
							(*ParameterType:=ParameterType,*) Axis:= Axis, ValueLreal:= lrValue, ValueDword := dwValue, ValueBool := bValue,
							ParameterPointer := ParameterPointer, ParameterSize:=ParameterSize); 
		state:=state + 1;
	END_IF;
	
	1 :	
	fbReadWriteParameter(Axis:= Axis, ValueLreal:= lrValue, ValueDword := dwValue, ValueBool := bValue);
	IF fbReadWriteParameter.Done THEN
		fbReadWriteParameter(Enable:= FALSE, ParameterNumber:= iParameterNumber, Mode:= READWRITEPARAMETERMODE_WRITE,
						(*ParameterType:= ParameterType,*) Axis:= Axis, ValueLreal:= lrValue, ValueDword := dwValue, ValueBool := bValue);
		state:=state + 1;
	END_IF;
	IF fbReadWriteParameter.Error THEN
		Busy := FALSE;
		Done := FALSE;
		Error := TRUE;
		ErrorID := fbReadWriteParameter.ErrorID;
		fbReadWriteParameter(Enable:= FALSE, ParameterNumber:= iParameterNumber, Mode:= READWRITEPARAMETERMODE_WRITE,
						(*ParameterType:= ParameterType,*) Axis:= Axis, ValueLreal:= lrValue, ValueDword := dwValue, ValueBool := bValue);
		state:=0;
	END_IF;
	
	2 : // write persistent parameter
	stParaStruct := _F_GetIndexGroup(ParaNumber := iParameterNumber, ControlLoopIndex := Axis.NcToPlc.ControlLoopIndex, Mode:=READWRITEPARAMETERMODE_WRITE);
	IG := stParaStruct.IndexGroup + Axis.NcToPlc.AxisId;	// Index Group of parameter		
	IO := stParaStruct.IndexOffset;							// Index Offset of parameter
	sTmp := _F_TcMC_DWORD_TO_HEXSTR2(IG, 4, TRUE);	
	sKey := CONCAT('NC: ChangeParameter ', sTmp);
	sTmp := _F_TcMC_DWORD_TO_HEXSTR2(IO, 8, TRUE);
	sKey := CONCAT(sKey, sTmp);								// unique ID string that describes the boot parameter 
//	sMsg := CONCAT('Initialization of boot parameter failed (MC_WriteParameterPersistent), ', sKey); 	// Logger string in case of initialization failure - added 20150623 KSt
	sMsg := 'Initialization of boot parameter failed (MC_WriteParameterPersistent)'; 	// Logger string in case of initialization failure - added 20150623 KSt
//	size := INT_TO_UINT( SIZEOF(AdsAddInitCommand) + LEN(sKey) + 1 + LEN(sMsg) + 1 + 
//						 SEL( ParameterType=PARAMETERTYPE_BOOL, SIZEOF(Value), SIZEOF(bValueWord) ) );	// complete length of command to SystemService
	CASE stParaStruct.ParaType OF	(* 2018-11-22 KSt *)
		PARAMETERTYPE_BOOL :	valuesize := SIZEOF(bValueWord);
		PARAMETERTYPE_DWORD:	valuesize := SIZEOF(dwValue);
		PARAMETERTYPE_LREAL:	valuesize := SIZEOF(lrValue);
		PARAMETERTYPE_LARGE: 	valuesize := ParameterSize;// for structured parameters  - KSt 2021-03-04
	ELSE
		valuesize := SIZEOF(lrValue);
	END_CASE

	size := valuesize + SIZEOF(AdsAddInitCommand) + INT_TO_UINT(LEN(sKey)) + 1 + INT_TO_UINT(LEN(sMsg)) + 1; // complete length of command to SystemService
	pCmd := ADR(aCmdBuffer);
		memset(pCmd, 0, size);	// initialize memory with zero bytes
		pCmd^.addr.port := 500;	// initialise AdsAddInitCommand structure
		pCmd^.initNo := 34;		// defined INIT constant for this function - don't change
		pCmd^.indexGroup := IG;
		pCmd^.indexOffset := IO;
		pCmd^.keyLength := INT_TO_UINT(LEN(sKey));
		pCmd^.msgLength := INT_TO_UINT(LEN(sMsg));
//		pCmd^.dataLength := SEL( ParameterType=PARAMETERTYPE_BOOL, SIZEOF(Value), SIZEOF(bValueWord));
		pCmd^.dataLength := valuesize;
		pCmd^.timeout := 0;
		pByte := pCmd + SIZEOF(AdsAddInitCommand);			// set pointer behind AdsAddInitCommand
		memcpy(pByte, ADR(sKey), INT_TO_UINT(LEN(sKey)));	// copy sKey string into structure
		pByte := pByte + INT_TO_UINT(LEN(sKey)) + 1;		// set pointer behind zero terminated string sKey
		memcpy(pByte, ADR(sMsg), INT_TO_UINT(LEN(sMsg)));	// copy sMsg (logger message) into structure 
		pByte := pByte + INT_TO_UINT(LEN(sMsg)) + 1;		// set pointer behind zero terminated string sMsg		
//		IF ParameterType=PARAMETERTYPE_BOOL THEN
//			memcpy(pByte, ADR(bValueWord), SIZEOF(bValueWord));	// copy parameter data (here 1 BOOL as UINT) into structure
//		ELSE
//			memcpy(pByte, ADR(Value), SIZEOF(Value));		// copy parameter data (here 1 LREAL) into structure
//		END_IF*)
		CASE stParaStruct.ParaType OF	(* 2018-11-22 KSt *)
			PARAMETERTYPE_BOOL :	memcpy(pByte, ADR(bValueWord), SIZEOF(bValueWord));
			PARAMETERTYPE_DWORD:	memcpy(pByte, ADR(dwValue), SIZEOF(dwValue));
			PARAMETERTYPE_LREAL:	memcpy(pByte, ADR(lrValue), SIZEOF(lrValue));
			PARAMETERTYPE_LARGE:	memcpy(pByte, ParameterPointer, ParameterSize);// for structured parameters  - KSt 2021-03-04
		ELSE
			memcpy(pByte, ADR(lrValue), SIZEOF(lrValue));
		END_CASE
		pByte := 0;											
		fbAdsWriteSystemService(PORT:=10000, IDXGRP:=170, IDXOFFS:=0, SRCADDR:=pCmd, LEN:=size, WRITE:=TRUE);	// send command to System Service
		state := state + 1;
	
	3 :
	fbAdsWriteSystemService();
	IF NOT fbAdsWriteSystemService.BUSY THEN
		Error := fbAdsWriteSystemService.ERR;
		ErrorID := fbAdsWriteSystemService.ERRID;
		Done := NOT Error;
		fbAdsWriteSystemService( WRITE:=FALSE );
		state := 0;
	END_IF
END_CASE

IF state=0 THEN
	Busy := FALSE;
END_IF
ADSbusy := fbReadWriteParameter.ADSbusy OR fbAdsWriteSystemService.BUSY;

END_FUNCTION_BLOCK

// POUs/Administrative/Status and Parameter/MC_WriteParameter
FUNCTION_BLOCK MC_WriteParameter
(*	This Function Block modifies the value of a vendor specific parameter. *)
VAR_IN_OUT
	Axis				:	AXIS_REF; (*Reference to an axis*)
END_VAR
VAR_INPUT
	Execute			:	BOOL;	
	ParameterNumber	:	MC_AxisParameter; // 2023-03 KSt changed from INT to MC_AxisParameter		
	Value			:	LREAL;	
(* 	ExecutionMode 	: 	MC_EXECUTION_MODE *)	(* not available *)
END_VAR
VAR_OUTPUT
	Done			:	BOOL;		
	Busy			: 	BOOL;		
	Error			:	BOOL;		
{attribute 'displaymode':='hex'}
	ErrorID			:	UDINT;		
END_VAR
VAR
	ADSbusy		: 	BOOL;
	fbReadWriteParameter: _FB_ReadWriteParameter;
END_VAR
VAR
//{attribute 'conditionalshow'}
//	nParatype 		:	_E_ParameterType;	(* removed 2021-04-12 KSt - not required *)
{attribute 'conditionalshow'}
	dwValue 			: 	DWORD;
{attribute 'conditionalshow'}
	bValue 			: 	BOOL;
{attribute 'conditionalshow'}
	fbTrigger 		: 	R_TRIG;
END_VAR

IF NOT Execute THEN
	Done := FALSE;
	Error := FALSE;			(* reset at falling edge of Execute *)
	ErrorID := 0;
END_IF
fbTrigger(CLK:= Execute);
IF fbTrigger.Q AND NOT Busy THEN
	Busy := TRUE;
	Done := FALSE;
	Error := FALSE;
	ErrorID := MC_ERROR_NO_ERROR;
END_IF;
(* *)
IF Busy THEN
//	nParatype := PARAMETERTYPE_LREAL;
	fbReadWriteParameter.ParameterPointer := 0;
	fbReadWriteParameter.ParameterSize := 0;
	bValue := Value<>0; (* 2010-05-04 KST - to write bool parameters with MC_WriteParameter as well *)
	fbReadWriteParameter(Enable:= TRUE, ParameterNumber:= ParameterNumber, Mode:= READWRITEPARAMETERMODE_WRITE,
						(*ParameterType:=nParatype,*) Axis:= Axis, ValueLreal:= Value, ValueDword := dwValue, ValueBool := bValue);
	IF fbReadWriteParameter.Done THEN
		Done := TRUE;
		Busy := FALSE;
		fbReadWriteParameter(Enable:= FALSE, ParameterNumber:= ParameterNumber, Mode:= READWRITEPARAMETERMODE_WRITE,
						(*ParameterType:= nParatype,*) Axis:= Axis, ValueLreal:= Value, ValueDword := dwValue, ValueBool := bValue);
	END_IF;
	IF fbReadWriteParameter.Error THEN
		Busy := FALSE;
		Done := FALSE;
		Error := TRUE;
		ErrorID := fbReadWriteParameter.ErrorID;
		fbReadWriteParameter(Enable:= FALSE, ParameterNumber:= ParameterNumber, Mode:= READWRITEPARAMETERMODE_WRITE,
						(*ParameterType:= nParatype,*) Axis:= Axis, ValueLreal:= Value, ValueDword := dwValue, ValueBool := bValue);
	END_IF;
END_IF;

ADSbusy := fbReadWriteParameter.ADSbusy;

END_FUNCTION_BLOCK

// POUs/Administrative/Status and Parameter/MC_WriteParameterPersistent
FUNCTION_BLOCK MC_WriteParameterPersistent
VAR_IN_OUT
	Axis: AXIS_REF; (*Reference to an axis*)
END_VAR
VAR_INPUT
	Execute: BOOL;
	ParameterNumber: MC_AxisParameter; // 2023-03 KSt changed from INT to MC_AxisParameter
	Value: LREAL;
END_VAR
VAR_OUTPUT
	Done: BOOL;
	Busy: BOOL;
	Error: BOOL;
{attribute 'displaymode':='hex'}
	ErrorID: UDINT;
END_VAR
VAR
	fbWriteParameterPersistent: _FB_WriteParameterPersistent;
END_VAR

fbWriteParameterPersistent(
	Axis:= Axis, 
	Execute:= Execute, 
	ParameterNumber:= ParameterNumber, 
	Value:= Value, 
//	ParameterType:= PARAMETERTYPE_LREAL, 	(* removed 2018-11-22 KSt - not required *)
	Done=> Done, 
	Busy=> Busy, 
	Error=> Error, 
	ErrorID=> ErrorID);

END_FUNCTION_BLOCK

// POUs/[obsolete]/F_GetVersion_TcMC2
{attribute 'hide'}
{attribute 'obsolete' := 'F_GetVersion_TcMC2 is obsolete, use stLibVersion_Tc2_MC2 instead!'}
FUNCTION F_GetVersion_TcMC2 : UINT	(* Gets the library version info *)
VAR_INPUT
	nVersionElement		:	INT;
END_VAR
(*
	Possible nVersionElement parameter:
	1	:	major number
	2	:	minor number
	3	:	revision number
*)

